LIN {X 0,Y 159.635,Z 839.585,A -85,B 0,C 180,E1 -24712.11,E2 -24712.11} C_VEL
LIN {X 0,Y 158.512,Z 849.666,A -85,B 0,C 180,E1 -24712.886,E2 -24712.886} C_VEL
LIN {X 0,Y 156.369,Z 861.365,A -85,B 0,C 180,E1 -24714.248,E2 -24714.248} C_VEL
LIN {X 0,Y 154.242,Z 870.146,A -85,B 0,C 180,E1 -24715.676,E2 -24715.676} C_VEL
LIN {X 0,Y 151.874,Z 878.505,A -85,B 0,C 180,E1 -24717.456,E2 -24717.456} C_VEL
LIN {X 0,Y 149.469,Z 885.387,A -85,B 0,C 180,E1 -24719.247,E2 -24719.247} C_VEL
LIN {X 0,Y 146.966,Z 892.073,A -85,B 0,C 180,E1 -24721.432,E2 -24721.432} C_VEL
LIN {X 0,Y 144.263,Z 898.407,A -85,B 0,C 180,E1 -24723.995,E2 -24723.995} C_VEL
LIN {X 0,Y 141.947,Z 903.667,A -85,B 0,C 180,E1 -24726.666,E2 -24726.666} C_VEL
LIN {X 0,Y 139.836,Z 908.059,A -85,B 0,C 180,E1 -24729.402,E2 -24729.402} C_VEL
LIN {X 0,Y 137.318,Z 913.221,A -85,B 0,C 180,E1 -24733.651,E2 -24733.651} C_VEL
LIN {X 0,Y 136.014,Z 915.865,A -85,B 0,C 180,E1 -24736.554,E2 -24736.554} C_VEL
LIN {X 0,Y 134.612,Z 918.759,A -85,B 0,C 180,E1 -24740.989,E2 -24740.989} C_VEL
LIN {X 0,Y 134.025,Z 920.018,A -85,B 0,C 180,E1 -24743.98,E2 -24743.98} C_VEL
LIN {X 0,Y 133.644,Z 920.881,A -85,B 0,C 180,E1 -24747.665,E2 -24747.665} C_VEL
LIN {X 0,Y 133.579,Z 920.989,A -85,B 0,C 180,E1 -24751.506,E2 -24751.506} C_VEL
LIN {X 0,Y 134.025,Z 920.078,A -85,B 0,C 180,E1 -24756.02,E2 -24756.02} C_VEL
LIN {X 0,Y 134.605,Z 918.859,A -85,B 0,C 180,E1 -24759.012,E2 -24759.012} C_VEL
LIN {X 0,Y 135.974,Z 916.007,A -85,B 0,C 180,E1 -24763.45,E2 -24763.45} C_VEL
LIN {X 0,Y 137.259,Z 913.408,A -85,B 0,C 180,E1 -24766.356,E2 -24766.356} C_VEL
LIN {X 0,Y 139.777,Z 908.296,A -85,B 0,C 180,E1 -24770.607,E2 -24770.607} C_VEL
LIN {X 0,Y 142.479,Z 902.79,A -85,B 0,C 180,E1 -24774.013,E2 -24774.013} C_VEL
LIN {X 0,Y 145.543,Z 895.866,A -85,B 0,C 180,E1 -24777.306,E2 -24777.306} C_VEL
LIN {X 0,Y 148.7,Z 887.912,A -85,B 0,C 180,E1 -24780.144,E2 -24780.144} C_VEL
LIN {X 0,Y 151.398,Z 880.327,A -85,B 0,C 180,E1 -24782.265,E2 -24782.265} C_VEL
LIN {X 0,Y 153.812,Z 872.37,A -85,B 0,C 180,E1 -24784.037,E2 -24784.037} C_VEL
LIN {X 0,Y 155.916,Z 864.14,A -85,B 0,C 180,E1 -24785.475,E2 -24785.475} C_VEL
LIN {X 0,Y 157.792,Z 855.078,A -85,B 0,C 180,E1 -24786.679,E2 -24786.679} C_VEL
LIN {X 0,Y 159.073,Z 846.352,A -85,B 0,C 180,E1 -24787.55,E2 -24787.55} C_VEL
LIN {X 0,Y 159.964,Z 837.426,A -85,B 0,C 180,E1 -24788.159,E2 -24788.159} C_VEL
LIN {X 0,Y 161.274,Z 812.923,A -85,B 0,C 180,E1 -24789.231,E2 -24789.231} C_VEL
LIN {X 0,Y 158.219,Z 805.845,A -85,B 0,C 180,E1 -24790.561,E2 -24790.561} C_VEL
LIN {X 0,Y 151.819,Z 794.198,A -85,B 0,C 180,E1 -24793.417,E2 -24793.417} C_VEL
LIN {X 0,Y 146.722,Z 786.269,A -85,B 0,C 180,E1 -24795.889,E2 -24795.889} C_VEL
LIN {X 0,Y 144.688,Z 783.348,A -85,B 0,C 180,E1 -24796.94,E2 -24796.94} C_VEL
LIN {X 0,Y 142.122,Z 779.603,A -85,B 0,C 180,E1 -24798.345,E2 -24798.345} C_VEL
LIN {X 0,Y 139.81,Z 776.247,A -85,B 0,C 180,E1 -24799.69,E2 -24799.69} C_VEL
LIN {X 0,Y 139.073,Z 775.314,A -85,B 0,C 180,E1 -24800.125,E2 -24800.125} C_VEL
LIN {X 0,Y 136.97,Z 773.087,A -85,B 0,C 180,E1 -24801.381,E2 -24801.381} C_VEL
LIN {X 0,Y 136.153,Z 770.959,A -85,B 0,C 180,E1 -24802.195,E2 -24802.195} C_VEL
LIN {X 0,Y 136.027,Z 770.381,A -85,B 0,C 180,E1 -24803.085,E2 -24803.085} C_VEL
LIN {X 0,Y 136.063,Z 770.334,A -85,B 0,C 180,E1 -24808.9,E2 -24808.9} C_VEL
LIN {X 0,Y 136.145,Z 770.314,A -85,B 0,C 180,E1 -24812.316,E2 -24812.316} C_VEL
LIN {X 0,Y 136.243,Z 770.325,A -85,B 0,C 180,E1 -24818.832,E2 -24818.832} C_VEL
LIN {X 0,Y 136.264,Z 770.295,A -85,B 0,C 180,E1 -24825.055,E2 -24825.055} C_VEL
LIN {X 0,Y 136.498,Z 770.293,A -85,B 0,C 180,E1 -24828.114,E2 -24828.114} C_VEL
LIN {X 0,Y 136.596,Z 770.241,A -85,B 0,C 180,E1 -24831.12,E2 -24831.12} C_VEL
LIN {X 0,Y 137.135,Z 770.182,A -85,B 0,C 180,E1 -24840,E2 -24840} C_VEL
LIN {X 0,Y 136.59,Z 770.268,A -85,B 0,C 180,E1 -24848.879,E2 -24848.879} C_VEL
LIN {X 0,Y 136.492,Z 770.252,A -85,B 0,C 180,E1 -24851.954,E2 -24851.954} C_VEL
LIN {X 0,Y 136.252,Z 770.315,A -85,B 0,C 180,E1 -24858.028,E2 -24858.028} C_VEL
LIN {X 0,Y 136.199,Z 770.294,A -85,B 0,C 180,E1 -24861.749,E2 -24861.749} C_VEL
LIN {X 0,Y 136.1,Z 770.315,A -85,B 0,C 180,E1 -24868.615,E2 -24868.615} C_VEL
LIN {X 0,Y 136.072,Z 770.314,A -85,B 0,C 180,E1 -24874.62,E2 -24874.62} C_VEL
LIN {X 0,Y 136.069,Z 770.603,A -85,B 0,C 180,E1 -24877.074,E2 -24877.074} C_VEL
LIN {X 0,Y 136.331,Z 771.59,A -85,B 0,C 180,E1 -24877.746,E2 -24877.746} C_VEL
LIN {X 0,Y 137.768,Z 774.133,A -85,B 0,C 180,E1 -24878.751,E2 -24878.751} C_VEL
LIN {X 0,Y 139.692,Z 775.951,A -85,B 0,C 180,E1 -24879.861,E2 -24879.861} C_VEL
LIN {X 0,Y 141.889,Z 779.358,A -85,B 0,C 180,E1 -24881.161,E2 -24881.161} C_VEL
LIN {X 0,Y 143.184,Z 781.06,A -85,B 0,C 180,E1 -24881.872,E2 -24881.872} C_VEL
LIN {X 0,Y 146.021,Z 785.342,A -85,B 0,C 180,E1 -24883.391,E2 -24883.391} C_VEL
LIN {X 0,Y 150.796,Z 794.191,A -85,B 0,C 180,E1 -24885.843,E2 -24885.843} C_VEL
LIN {X 0,Y 155.885,Z 805.497,A -85,B 0,C 180,E1 -24888.306,E2 -24888.306} C_VEL
LIN {X 0,Y 159.778,Z 815.797,A -85,B 0,C 180,E1 -24890.122,E2 -24890.122} C_VEL
LIN {X 0,Y 160.657,Z 825.932,A -85,B 0,C 180,E1 -24890.954,E2 -24890.954} C_VEL
LIN {X 0,Y 159.375,Z 846.828,A -85,B 0,C 180,E1 -24891.876,E2 -24891.876} C_VEL
LIN {X 0,Y 157.91,Z 858.37,A -85,B 0,C 180,E1 -24892.735,E2 -24892.735} C_VEL
LIN {X 0,Y 155.604,Z 869.497,A -85,B 0,C 180,E1 -24894.044,E2 -24894.044} C_VEL
LIN {X 0,Y 153.331,Z 878.512,A -85,B 0,C 180,E1 -24895.535,E2 -24895.535} C_VEL
LIN {X 0,Y 150.925,Z 886.424,A -85,B 0,C 180,E1 -24897.215,E2 -24897.215} C_VEL
LIN {X 0,Y 148.126,Z 894.308,A -85,B 0,C 180,E1 -24899.333,E2 -24899.333} C_VEL
LIN {X 0,Y 145.178,Z 901.651,A -85,B 0,C 180,E1 -24901.836,E2 -24901.836} C_VEL
LIN {X 0,Y 141.973,Z 909.104,A -85,B 0,C 180,E1 -24905.117,E2 -24905.117} C_VEL
LIN {X 0,Y 139.22,Z 914.946,A -85,B 0,C 180,E1 -24908.532,E2 -24908.532} C_VEL
LIN {X 0,Y 137.076,Z 919.559,A -85,B 0,C 180,E1 -24912.084,E2 -24912.084} C_VEL
LIN {X 0,Y 135.739,Z 922.56,A -85,B 0,C 180,E1 -24914.996,E2 -24914.996} C_VEL
LIN {X 0,Y 134.718,Z 924.892,A -85,B 0,C 180,E1 -24917.955,E2 -24917.955} C_VEL
LIN {X 0,Y 133.989,Z 926.641,A -85,B 0,C 180,E1 -24920.947,E2 -24920.947} C_VEL
LIN {X 0,Y 133.631,Z 927.895,A -85,B 0,C 180,E1 -24923.962,E2 -24923.962} C_VEL
LIN {X 0,Y 133.47,Z 928.674,A -85,B 0,C 180,E1 -24926.982,E2 -24926.982} C_VEL
LIN {X 0,Y 133.531,Z 928.971,A -85,B 0,C 180,E1 -24930,E2 -24930} C_VEL
LIN {X 0,Y 133.467,Z 928.664,A -85,B 0,C 180,E1 -24933.018,E2 -24933.018} C_VEL
LIN {X 0,Y 133.571,Z 927.863,A -85,B 0,C 180,E1 -24936.041,E2 -24936.041} C_VEL
LIN {X 0,Y 133.989,Z 926.589,A -85,B 0,C 180,E1 -24939.053,E2 -24939.053} C_VEL
LIN {X 0,Y 135.186,Z 923.659,A -85,B 0,C 180,E1 -24943.529,E2 -24943.529} C_VEL
LIN {X 0,Y 136.362,Z 920.99,A -85,B 0,C 180,E1 -24946.467,E2 -24946.467} C_VEL
LIN {X 0,Y 138.728,Z 915.782,A -85,B 0,C 180,E1 -24950.77,E2 -24950.77} C_VEL
LIN {X 0,Y 141.96,Z 908.923,A -85,B 0,C 180,E1 -24954.886,E2 -24954.886} C_VEL
LIN {X 0,Y 145.158,Z 901.434,A -85,B 0,C 180,E1 -24958.168,E2 -24958.168} C_VEL
LIN {X 0,Y 148.13,Z 894.053,A -85,B 0,C 180,E1 -24960.666,E2 -24960.666} C_VEL
LIN {X 0,Y 148.755,Z 892.384,A -85,B 0,C 180,E1 -24961.166,E2 -24961.166} C_VEL
LIN {X 0,Y 149.828,Z 887.833,A -85,B 0,C 180,E1 -24962.562,E2 -24962.562} C_VEL
LIN {X 0,Y 149.907,Z 880.057,A -85,B 0,C 180,E1 -24964.93,E2 -24964.93} C_VEL
LIN {X 0,Y 149.788,Z 871.747,A -85,B 0,C 180,E1 -24967.002,E2 -24967.002} C_VEL
LIN {X 0,Y 150.487,Z 866.362,A -85,B 0,C 180,E1 -24967.892,E2 -24967.892} C_VEL
LIN {X 0,Y 152.584,Z 855.455,A -85,B 0,C 180,E1 -24969.045,E2 -24969.045} C_VEL
LIN {X 0,Y 153.775,Z 846.031,A -85,B 0,C 180,E1 -24969.717,E2 -24969.717} C_VEL
LIN {X 0,Y 154.965,Z 825.846,A -85,B 0,C 180,E1 -24970.654,E2 -24970.654} C_VEL
LIN {X 0,Y 154.102,Z 817.408,A -85,B 0,C 180,E1 -24971.438,E2 -24971.438} C_VEL
LIN {X 0,Y 149.667,Z 805.878,A -85,B 0,C 180,E1 -24973.685,E2 -24973.685} C_VEL
LIN {X 0,Y 145.152,Z 796.052,A -85,B 0,C 180,E1 -24976.078,E2 -24976.078} C_VEL
LIN {X 0,Y 141.174,Z 788.802,A -85,B 0,C 180,E1 -24978.304,E2 -24978.304} C_VEL
LIN {X 0,Y 138.212,Z 784.573,A -85,B 0,C 180,E1 -24980.023,E2 -24980.023} C_VEL
LIN {X 0,Y 135.846,Z 781.103,A -85,B 0,C 180,E1 -24981.505,E2 -24981.505} C_VEL
LIN {X 0,Y 133.439,Z 778.063,A -85,B 0,C 180,E1 -24983.077,E2 -24983.077} C_VEL
LIN {X 0,Y 132.663,Z 776.576,A -85,B 0,C 180,E1 -24983.653,E2 -24983.653} C_VEL
LIN {X 0,Y 130.343,Z 774.52,A -85,B 0,C 180,E1 -24985.244,E2 -24985.244} C_VEL
LIN {X 0,Y 129.107,Z 771.819,A -85,B 0,C 180,E1 -24986.543,E2 -24986.543} C_VEL
LIN {X 0,Y 128.986,Z 771.241,A -85,B 0,C 180,E1 -24987.911,E2 -24987.911} C_VEL
LIN {X 0,Y 129.017,Z 771.195,A -85,B 0,C 180,E1 -24990.643,E2 -24990.643} C_VEL
LIN {X 0,Y 129.031,Z 771.225,A -85,B 0,C 180,E1 -24994.168,E2 -24994.168} C_VEL
LIN {X 0,Y 129.108,Z 771.178,A -85,B 0,C 180,E1 -24997.728,E2 -24997.728} C_VEL
LIN {X 0,Y 129.159,Z 771.183,A -85,B 0,C 180,E1 -25000.945,E2 -25000.945} C_VEL
LIN {X 0,Y 129.417,Z 771.132,A -85,B 0,C 180,E1 -25007.821,E2 -25007.821} C_VEL
LIN {X 0,Y 129.516,Z 771.14,A -85,B 0,C 180,E1 -25010.631,E2 -25010.631} C_VEL
LIN {X 0,Y 130.091,Z 771.058,A -85,B 0,C 180,E1 -25020,E2 -25020} C_VEL
LIN {X 0,Y 129.511,Z 771.125,A -85,B 0,C 180,E1 -25029.37,E2 -25029.37} C_VEL
LIN {X 0,Y 129.392,Z 771.181,A -85,B 0,C 180,E1 -25032.549,E2 -25032.549} C_VEL
LIN {X 0,Y 129.114,Z 771.181,A -85,B 0,C 180,E1 -25039.063,E2 -25039.063} C_VEL
LIN {X 0,Y 129.107,Z 771.209,A -85,B 0,C 180,E1 -25042.399,E2 -25042.399} C_VEL
LIN {X 0,Y 129.027,Z 771.19,A -85,B 0,C 180,E1 -25045.834,E2 -25045.834} C_VEL
LIN {X 0,Y 129.017,Z 771.221,A -85,B 0,C 180,E1 -25049.358,E2 -25049.358} C_VEL
LIN {X 0,Y 129.033,Z 771.485,A -85,B 0,C 180,E1 -25053.534,E2 -25053.534} C_VEL
LIN {X 0,Y 129.324,Z 772.589,A -85,B 0,C 180,E1 -25054.339,E2 -25054.339} C_VEL
LIN {X 0,Y 130.811,Z 775.152,A -85,B 0,C 180,E1 -25055.566,E2 -25055.566} C_VEL
LIN {X 0,Y 132.899,Z 777.009,A -85,B 0,C 180,E1 -25056.981,E2 -25056.981} C_VEL
LIN {X 0,Y 134.985,Z 780.287,A -85,B 0,C 180,E1 -25058.428,E2 -25058.428} C_VEL
LIN {X 0,Y 136.568,Z 782.116,A -85,B 0,C 180,E1 -25059.413,E2 -25059.413} C_VEL
LIN {X 0,Y 140.219,Z 787.446,A -85,B 0,C 180,E1 -25061.616,E2 -25061.616} C_VEL
LIN {X 0,Y 145.335,Z 795.26,A -85,B 0,C 180,E1 -25064.401,E2 -25064.401} C_VEL
LIN {X 0,Y 150.635,Z 804.437,A -85,B 0,C 180,E1 -25067.03,E2 -25067.03} C_VEL
LIN {X 0,Y 155.264,Z 813.871,A -85,B 0,C 180,E1 -25069.183,E2 -25069.183} C_VEL
LIN {X 0,Y 155.734,Z 815.756,A -85,B 0,C 180,E1 -25069.446,E2 -25069.446} C_VEL
LIN {X 0,Y 154.175,Z 838.958,A -85,B 0,C 180,E1 -25070.444,E2 -25070.444} C_VEL
LIN {X 0,Y 153.149,Z 848.227,A -85,B 0,C 180,E1 -25071.142,E2 -25071.142} C_VEL
LIN {X 0,Y 151.218,Z 859.169,A -85,B 0,C 180,E1 -25072.327,E2 -25072.327} C_VEL
LIN {X 0,Y 148.44,Z 870.36,A -85,B 0,C 180,E1 -25074.133,E2 -25074.133} C_VEL
LIN {X 0,Y 145.938,Z 878.718,A -85,B 0,C 180,E1 -25075.956,E2 -25075.956} C_VEL
LIN {X 0,Y 143.431,Z 885.598,A -85,B 0,C 180,E1 -25077.801,E2 -25077.801} C_VEL
LIN {X 0,Y 140.791,Z 892.284,A -85,B 0,C 180,E1 -25080.054,E2 -25080.054} C_VEL
LIN {X 0,Y 137.919,Z 898.618,A -85,B 0,C 180,E1 -25082.702,E2 -25082.702} C_VEL
LIN {X 0,Y 135.455,Z 903.878,A -85,B 0,C 180,E1 -25085.476,E2 -25085.476} C_VEL
LIN {X 0,Y 133.214,Z 908.269,A -85,B 0,C 180,E1 -25088.327,E2 -25088.327} C_VEL
LIN {X 0,Y 130.531,Z 913.431,A -85,B 0,C 180,E1 -25092.775,E2 -25092.775} C_VEL
LIN {X 0,Y 129.118,Z 916.075,A -85,B 0,C 180,E1 -25095.822,E2 -25095.822} C_VEL
LIN {X 0,Y 127.614,Z 918.969,A -85,B 0,C 180,E1 -25100.49,E2 -25100.49} C_VEL
LIN {X 0,Y 126.971,Z 920.228,A -85,B 0,C 180,E1 -25103.644,E2 -25103.644} C_VEL
LIN {X 0,Y 126.617,Z 921.018,A -85,B 0,C 180,E1 -25106.818,E2 -25106.818} C_VEL
LIN {X 0,Y 126.505,Z 921.319,A -85,B 0,C 180,E1 -25110,E2 -25110} C_VEL
LIN {X 0,Y 126.586,Z 921.039,A -85,B 0,C 180,E1 -25113.183,E2 -25113.183} C_VEL
LIN {X 0,Y 126.971,Z 920.286,A -85,B 0,C 180,E1 -25116.356,E2 -25116.356} C_VEL
LIN {X 0,Y 127.607,Z 919.068,A -85,B 0,C 180,E1 -25119.51,E2 -25119.51} C_VEL
LIN {X 0,Y 129.08,Z 916.215,A -85,B 0,C 180,E1 -25124.183,E2 -25124.183} C_VEL
LIN {X 0,Y 130.464,Z 913.616,A -85,B 0,C 180,E1 -25127.234,E2 -25127.234} C_VEL
LIN {X 0,Y 133.16,Z 908.503,A -85,B 0,C 180,E1 -25131.682,E2 -25131.682} C_VEL
LIN {X 0,Y 136.034,Z 902.997,A -85,B 0,C 180,E1 -25135.228,E2 -25135.228} C_VEL
LIN {X 0,Y 139.279,Z 896.072,A -85,B 0,C 180,E1 -25138.644,E2 -25138.644} C_VEL
LIN {X 0,Y 142.625,Z 888.117,A -85,B 0,C 180,E1 -25141.571,E2 -25141.571} C_VEL
LIN {X 0,Y 145.454,Z 880.531,A -85,B 0,C 180,E1 -25143.756,E2 -25143.756} C_VEL
LIN {X 0,Y 147.993,Z 872.574,A -85,B 0,C 180,E1 -25145.573,E2 -25145.573} C_VEL
LIN {X 0,Y 150.213,Z 864.342,A -85,B 0,C 180,E1 -25147.041,E2 -25147.041} C_VEL
LIN {X 0,Y 152.093,Z 855.662,A -85,B 0,C 180,E1 -25148.228,E2 -25148.228} C_VEL
LIN {X 0,Y 153.43,Z 847.101,A -85,B 0,C 180,E1 -25149.118,E2 -25149.118} C_VEL
LIN {X 0,Y 154.342,Z 838.914,A -85,B 0,C 180,E1 -25149.711,E2 -25149.711} C_VEL
LIN {X 0,Y 155.748,Z 814.926,A -85,B 0,C 180,E1 -25150.803,E2 -25150.803} C_VEL
LIN {X 0,Y 152.296,Z 807.458,A -85,B 0,C 180,E1 -25152.408,E2 -25152.408} C_VEL
LIN {X 0,Y 146.671,Z 797.355,A -85,B 0,C 180,E1 -25155.148,E2 -25155.148} C_VEL
LIN {X 0,Y 141.36,Z 789.057,A -85,B 0,C 180,E1 -25157.985,E2 -25157.985} C_VEL
LIN {X 0,Y 138.426,Z 784.813,A -85,B 0,C 180,E1 -25159.694,E2 -25159.694} C_VEL
LIN {X 0,Y 135.842,Z 781.12,A -85,B 0,C 180,E1 -25161.312,E2 -25161.312} C_VEL
LIN {X 0,Y 133.487,Z 778.201,A -85,B 0,C 180,E1 -25162.855,E2 -25162.855} C_VEL
LIN {X 0,Y 132.477,Z 776.49,A -85,B 0,C 180,E1 -25163.593,E2 -25163.593} C_VEL
LIN {X 0,Y 130.277,Z 774.484,A -85,B 0,C 180,E1 -25165.126,E2 -25165.126} C_VEL
LIN {X 0,Y 129.1,Z 771.782,A -85,B 0,C 180,E1 -25166.427,E2 -25166.427} C_VEL
LIN {X 0,Y 128.974,Z 771.233,A -85,B 0,C 180,E1 -25167.908,E2 -25167.908} C_VEL
LIN {X 0,Y 129.035,Z 771.221,A -85,B 0,C 180,E1 -25170.646,E2 -25170.646} C_VEL
LIN {X 0,Y 129.109,Z 771.207,A -85,B 0,C 180,E1 -25177.601,E2 -25177.601} C_VEL
LIN {X 0,Y 129.181,Z 771.169,A -85,B 0,C 180,E1 -25184.215,E2 -25184.215} C_VEL
LIN {X 0,Y 129.418,Z 771.177,A -85,B 0,C 180,E1 -25187.82,E2 -25187.82} C_VEL
LIN {X 0,Y 129.521,Z 771.125,A -85,B 0,C 180,E1 -25190.631,E2 -25190.631} C_VEL
LIN {X 0,Y 130.09,Z 771.059,A -85,B 0,C 180,E1 -25200,E2 -25200} C_VEL
LIN {X 0,Y 129.516,Z 771.14,A -85,B 0,C 180,E1 -25209.369,E2 -25209.369} C_VEL
LIN {X 0,Y 129.394,Z 771.135,A -85,B 0,C 180,E1 -25212.548,E2 -25212.548} C_VEL
LIN {X 0,Y 129.159,Z 771.183,A -85,B 0,C 180,E1 -25219.055,E2 -25219.055} C_VEL
LIN {X 0,Y 129.109,Z 771.179,A -85,B 0,C 180,E1 -25222.398,E2 -25222.398} C_VEL
LIN {X 0,Y 129.031,Z 771.225,A -85,B 0,C 180,E1 -25225.832,E2 -25225.832} C_VEL
LIN {X 0,Y 129.005,Z 771.255,A -85,B 0,C 180,E1 -25232.084,E2 -25232.084} C_VEL
LIN {X 0,Y 129.106,Z 771.784,A -85,B 0,C 180,E1 -25233.219,E2 -25233.219} C_VEL
LIN {X 0,Y 130.539,Z 774.745,A -85,B 0,C 180,E1 -25234.696,E2 -25234.696} C_VEL
LIN {X 0,Y 132.96,Z 777.036,A -85,B 0,C 180,E1 -25236.37,E2 -25236.37} C_VEL
LIN {X 0,Y 135.035,Z 780.3,A -85,B 0,C 180,E1 -25237.818,E2 -25237.818} C_VEL
LIN {X 0,Y 136.493,Z 781.884,A -85,B 0,C 180,E1 -25238.725,E2 -25238.725} C_VEL
LIN {X 0,Y 141.953,Z 789.956,A -85,B 0,C 180,E1 -25241.979,E2 -25241.979} C_VEL
LIN {X 0,Y 146.684,Z 799.062,A -85,B 0,C 180,E1 -25244.605,E2 -25244.605} C_VEL
LIN {X 0,Y 151.302,Z 809.666,A -85,B 0,C 180,E1 -25247.016,E2 -25247.016} C_VEL
LIN {X 0,Y 154.496,Z 818.541,A -85,B 0,C 180,E1 -25248.642,E2 -25248.642} C_VEL
LIN {X 0,Y 155.11,Z 827.574,A -85,B 0,C 180,E1 -25249.381,E2 -25249.381} C_VEL
LIN {X 0,Y 153.784,Z 847.481,A -85,B 0,C 180,E1 -25250.292,E2 -25250.292} C_VEL
LIN {X 0,Y 151.988,Z 859.859,A -85,B 0,C 180,E1 -25251.294,E2 -25251.294} C_VEL
LIN {X 0,Y 149.66,Z 870.325,A -85,B 0,C 180,E1 -25252.609,E2 -25252.609} C_VEL
LIN {X 0,Y 147.452,Z 878.55,A -85,B 0,C 180,E1 -25254.02,E2 -25254.02} C_VEL
LIN {X 0,Y 144.745,Z 886.981,A -85,B 0,C 180,E1 -25255.885,E2 -25255.885} C_VEL
LIN {X 0,Y 141.667,Z 895.125,A -85,B 0,C 180,E1 -25258.19,E2 -25258.19} C_VEL
LIN {X 0,Y 138.291,Z 903.144,A -85,B 0,C 180,E1 -25261.132,E2 -25261.132} C_VEL
LIN {X 0,Y 134.927,Z 910.138,A -85,B 0,C 180,E1 -25264.55,E2 -25264.55} C_VEL
LIN {X 0,Y 132.095,Z 915.699,A -85,B 0,C 180,E1 -25268.135,E2 -25268.135} C_VEL
LIN {X 0,Y 129.548,Z 920.878,A -85,B 0,C 180,E1 -25272.64,E2 -25272.64} C_VEL
LIN {X 0,Y 127.759,Z 924.684,A -85,B 0,C 180,E1 -25277.289,E2 -25277.289} C_VEL
LIN {X 0,Y 126.968,Z 926.432,A -85,B 0,C 180,E1 -25280.441,E2 -25280.441} C_VEL
LIN {X 0,Y 126.564,Z 927.687,A -85,B 0,C 180,E1 -25283.624,E2 -25283.624} C_VEL
LIN {X 0,Y 126.383,Z 928.466,A -85,B 0,C 180,E1 -25286.812,E2 -25286.812} C_VEL
LIN {X 0,Y 126.445,Z 928.762,A -85,B 0,C 180,E1 -25290,E2 -25290} C_VEL
LIN {X 0,Y 126.379,Z 928.455,A -85,B 0,C 180,E1 -25293.188,E2 -25293.188} C_VEL
LIN {X 0,Y 126.522,Z 927.654,A -85,B 0,C 180,E1 -25296.378,E2 -25296.378} C_VEL
LIN {X 0,Y 126.968,Z 926.379,A -85,B 0,C 180,E1 -25299.559,E2 -25299.559} C_VEL
LIN {X 0,Y 128.266,Z 923.448,A -85,B 0,C 180,E1 -25304.274,E2 -25304.274} C_VEL
LIN {X 0,Y 129.547,Z 920.779,A -85,B 0,C 180,E1 -25307.36,E2 -25307.36} C_VEL
LIN {X 0,Y 132.095,Z 915.571,A -85,B 0,C 180,E1 -25311.866,E2 -25311.866} C_VEL
LIN {X 0,Y 135.55,Z 908.712,A -85,B 0,C 180,E1 -25316.149,E2 -25316.149} C_VEL
LIN {X 0,Y 138.924,Z 901.222,A -85,B 0,C 180,E1 -25319.554,E2 -25319.554} C_VEL
LIN {X 0,Y 142.075,Z 893.841,A -85,B 0,C 180,E1 -25322.125,E2 -25322.125} C_VEL
LIN {X 0,Y 144.886,Z 886.228,A -85,B 0,C 180,E1 -25324.225,E2 -25324.225} C_VEL
LIN {X 0,Y 147.537,Z 877.723,A -85,B 0,C 180,E1 -25326.077,E2 -25326.077} C_VEL
LIN {X 0,Y 150.295,Z 867.26,A -85,B 0,C 180,E1 -25327.78,E2 -25327.78} C_VEL
LIN {X 0,Y 150.487,Z 866.362,A -85,B 0,C 180,E1 -25327.892,E2 -25327.892} C_VEL
LIN {X 0,Y 151.182,Z 860.851,A -85,B 0,C 180,E1 -25328.681,E2 -25328.681} C_VEL
LIN {X 0,Y 150.397,Z 851.78,A -85,B 0,C 180,E1 -25330.191,E2 -25330.191} C_VEL
LIN {X 0,Y 149.185,Z 842.523,A -85,B 0,C 180,E1 -25331.487,E2 -25331.487} C_VEL
LIN {X 0,Y 149.093,Z 836.717,A -85,B 0,C 180,E1 -25331.915,E2 -25331.915} C_VEL
LIN {X 0,Y 149.543,Z 826.064,A -85,B 0,C 180,E1 -25332.434,E2 -25332.434} C_VEL
LIN {X 0,Y 149.04,Z 820.348,A -85,B 0,C 180,E1 -25332.976,E2 -25332.976} C_VEL
LIN {X 0,Y 144.912,Z 809.373,A -85,B 0,C 180,E1 -25335.253,E2 -25335.253} C_VEL
LIN {X 0,Y 140.789,Z 800.186,A -85,B 0,C 180,E1 -25337.632,E2 -25337.632} C_VEL
LIN {X 0,Y 137.451,Z 793.945,A -85,B 0,C 180,E1 -25339.656,E2 -25339.656} C_VEL
LIN {X 0,Y 134.408,Z 789.463,A -85,B 0,C 180,E1 -25341.569,E2 -25341.569} C_VEL
LIN {X 0,Y 132.393,Z 786.53,A -85,B 0,C 180,E1 -25342.93,E2 -25342.93} C_VEL
LIN {X 0,Y 129.981,Z 783.042,A -85,B 0,C 180,E1 -25344.672,E2 -25344.672} C_VEL
LIN {X 0,Y 127.067,Z 779.637,A -85,B 0,C 180,E1 -25346.895,E2 -25346.895} C_VEL
LIN {X 0,Y 125.849,Z 777.609,A -85,B 0,C 180,E1 -25347.959,E2 -25347.959} C_VEL
LIN {X 0,Y 123.301,Z 775.404,A -85,B 0,C 180,E1 -25350.136,E2 -25350.136} C_VEL
LIN {X 0,Y 122.033,Z 772.697,A -85,B 0,C 180,E1 -25351.811,E2 -25351.811} C_VEL
LIN {X 0,Y 121.956,Z 772.124,A -85,B 0,C 180,E1 -25353.474,E2 -25353.474} C_VEL
LIN {X 0,Y 122.029,Z 772.063,A -85,B 0,C 180,E1 -25357.145,E2 -25357.145} C_VEL
LIN {X 0,Y 122.116,Z 772.085,A -85,B 0,C 180,E1 -25363.277,E2 -25363.277} C_VEL
LIN {X 0,Y 122.364,Z 772.01,A -85,B 0,C 180,E1 -25367.527,E2 -25367.527} C_VEL
LIN {X 0,Y 122.446,Z 772.013,A -85,B 0,C 180,E1 -25370.085,E2 -25370.085} C_VEL
LIN {X 0,Y 122.604,Z 771.978,A -85,B 0,C 180,E1 -25376.714,E2 -25376.714} C_VEL
LIN {X 0,Y 123.044,Z 771.935,A -85,B 0,C 180,E1 -25380,E2 -25380} C_VEL
LIN {X 0,Y 122.419,Z 772.001,A -85,B 0,C 180,E1 -25387.089,E2 -25387.089} C_VEL
LIN {X 0,Y 122.364,Z 772.056,A -85,B 0,C 180,E1 -25392.472,E2 -25392.472} C_VEL
LIN {X 0,Y 122.021,Z 772.076,A -85,B 0,C 180,E1 -25400.218,E2 -25400.218} C_VEL
LIN {X 0,Y 121.982,Z 772.077,A -85,B 0,C 180,E1 -25403.785,E2 -25403.785} C_VEL
LIN {X 0,Y 121.977,Z 772.402,A -85,B 0,C 180,E1 -25408.266,E2 -25408.266} C_VEL
LIN {X 0,Y 122.347,Z 773.615,A -85,B 0,C 180,E1 -25409.294,E2 -25409.294} C_VEL
LIN {X 0,Y 123.736,Z 776.07,A -85,B 0,C 180,E1 -25410.743,E2 -25410.743} C_VEL
LIN {X 0,Y 126.182,Z 777.945,A -85,B 0,C 180,E1 -25412.773,E2 -25412.773} C_VEL
LIN {X 0,Y 128.034,Z 781.091,A -85,B 0,C 180,E1 -25414.359,E2 -25414.359} C_VEL
LIN {X 0,Y 130.016,Z 783.198,A -85,B 0,C 180,E1 -25415.823,E2 -25415.823} C_VEL
LIN {X 0,Y 132.485,Z 786.66,A -85,B 0,C 180,E1 -25417.593,E2 -25417.593} C_VEL
LIN {X 0,Y 136.466,Z 792.391,A -85,B 0,C 180,E1 -25420.193,E2 -25420.193} C_VEL
LIN {X 0,Y 142.6,Z 802.122,A -85,B 0,C 180,E1 -25423.752,E2 -25423.752} C_VEL
LIN {X 0,Y 148.357,Z 813.011,A -85,B 0,C 180,E1 -25426.761,E2 -25426.761} C_VEL
LIN {X 0,Y 150.218,Z 816.904,A -85,B 0,C 180,E1 -25427.678,E2 -25427.678} C_VEL
LIN {X 0,Y 148.687,Z 840.407,A -85,B 0,C 180,E1 -25428.78,E2 -25428.78} C_VEL
LIN {X 0,Y 147.161,Z 852.138,A -85,B 0,C 180,E1 -25429.768,E2 -25429.768} C_VEL
LIN {X 0,Y 145.108,Z 861.794,A -85,B 0,C 180,E1 -25430.977,E2 -25430.977} C_VEL
LIN {X 0,Y 142.757,Z 870.573,A -85,B 0,C 180,E1 -25432.466,E2 -25432.466} C_VEL
LIN {X 0,Y 140.12,Z 878.93,A -85,B 0,C 180,E1 -25434.333,E2 -25434.333} C_VEL
LIN {X 0,Y 137.491,Z 885.81,A -85,B 0,C 180,E1 -25436.228,E2 -25436.228} C_VEL
LIN {X 0,Y 134.698,Z 892.495,A -85,B 0,C 180,E1 -25438.55,E2 -25438.55} C_VEL
LIN {X 0,Y 131.655,Z 898.829,A -85,B 0,C 180,E1 -25441.286,E2 -25441.286} C_VEL
LIN {X 0,Y 129.029,Z 904.088,A -85,B 0,C 180,E1 -25444.167,E2 -25444.167} C_VEL
LIN {X 0,Y 126.647,Z 908.479,A -85,B 0,C 180,E1 -25447.142,E2 -25447.142} C_VEL
LIN {X 0,Y 123.769,Z 913.641,A -85,B 0,C 180,E1 -25451.802,E2 -25451.802} C_VEL
LIN {X 0,Y 122.255,Z 916.285,A -85,B 0,C 180,E1 -25455.008,E2 -25455.008} C_VEL
LIN {X 0,Y 120.617,Z 919.178,A -85,B 0,C 180,E1 -25459.933,E2 -25459.933} C_VEL
LIN {X 0,Y 119.916,Z 920.437,A -85,B 0,C 180,E1 -25463.269,E2 -25463.269} C_VEL
LIN {X 0,Y 119.54,Z 921.227,A -85,B 0,C 180,E1 -25466.63,E2 -25466.63} C_VEL
LIN {X 0,Y 119.419,Z 921.528,A -85,B 0,C 180,E1 -25470,E2 -25470} C_VEL
LIN {X 0,Y 119.5,Z 921.247,A -85,B 0,C 180,E1 -25473.372,E2 -25473.372} C_VEL
LIN {X 0,Y 119.916,Z 920.495,A -85,B 0,C 180,E1 -25476.731,E2 -25476.731} C_VEL
LIN {X 0,Y 120.61,Z 919.276,A -85,B 0,C 180,E1 -25480.068,E2 -25480.068} C_VEL
LIN {X 0,Y 122.221,Z 916.423,A -85,B 0,C 180,E1 -25484.997,E2 -25484.997} C_VEL
LIN {X 0,Y 123.699,Z 913.823,A -85,B 0,C 180,E1 -25488.209,E2 -25488.209} C_VEL
LIN {X 0,Y 126.601,Z 908.71,A -85,B 0,C 180,E1 -25492.867,E2 -25492.867} C_VEL
LIN {X 0,Y 129.652,Z 903.204,A -85,B 0,C 180,E1 -25496.565,E2 -25496.565} C_VEL
LIN {X 0,Y 133.099,Z 896.278,A -85,B 0,C 180,E1 -25500.108,E2 -25500.108} C_VEL
LIN {X 0,Y 136.633,Z 888.323,A -85,B 0,C 180,E1 -25503.129,E2 -25503.129} C_VEL
LIN {X 0,Y 139.609,Z 880.736,A -85,B 0,C 180,E1 -25505.374,E2 -25505.374} C_VEL
LIN {X 0,Y 142.29,Z 872.777,A -85,B 0,C 180,E1 -25507.233,E2 -25507.233} C_VEL
LIN {X 0,Y 144.625,Z 864.544,A -85,B 0,C 180,E1 -25508.73,E2 -25508.73} C_VEL
LIN {X 0,Y 146.527,Z 856.163,A -85,B 0,C 180,E1 -25509.908,E2 -25509.908} C_VEL
LIN {X 0,Y 148.004,Z 847.266,A -85,B 0,C 180,E1 -25510.852,E2 -25510.852} C_VEL
LIN {X 0,Y 148.959,Z 839.107,A -85,B 0,C 180,E1 -25511.453,E2 -25511.453} C_VEL
LIN {X 0,Y 150.364,Z 817.143,A -85,B 0,C 180,E1 -25512.469,E2 -25512.469} C_VEL
LIN {X 0,Y 145.323,Z 806.897,A -85,B 0,C 180,E1 -25515.028,E2 -25515.028} C_VEL
LIN {X 0,Y 139.495,Z 796.988,A -85,B 0,C 180,E1 -25518.242,E2 -25518.242} C_VEL
LIN {X 0,Y 134.973,Z 790.201,A -85,B 0,C 180,E1 -25521.016,E2 -25521.016} C_VEL
LIN {X 0,Y 132.603,Z 786.76,A -85,B 0,C 180,E1 -25522.609,E2 -25522.609} C_VEL
LIN {X 0,Y 130.135,Z 783.36,A -85,B 0,C 180,E1 -25524.38,E2 -25524.38} C_VEL
LIN {X 0,Y 129.36,Z 782.368,A -85,B 0,C 180,E1 -25524.959,E2 -25524.959} C_VEL
LIN {X 0,Y 127.038,Z 779.658,A -85,B 0,C 180,E1 -25526.767,E2 -25526.767} C_VEL
LIN {X 0,Y 125.944,Z 777.662,A -85,B 0,C 180,E1 -25527.75,E2 -25527.75} C_VEL
LIN {X 0,Y 123.351,Z 775.485,A -85,B 0,C 180,E1 -25529.975,E2 -25529.975} C_VEL
LIN {X 0,Y 122.051,Z 772.712,A -85,B 0,C 180,E1 -25531.658,E2 -25531.658} C_VEL
LIN {X 0,Y 121.953,Z 772.111,A -85,B 0,C 180,E1 -25533.01,E2 -25533.01} C_VEL
LIN {X 0,Y 122.023,Z 772.082,A -85,B 0,C 180,E1 -25537.151,E2 -25537.151} C_VEL
LIN {X 0,Y 122.093,Z 772.047,A -85,B 0,C 180,E1 -25543.273,E2 -25543.273} C_VEL
LIN {X 0,Y 122.365,Z 772.056,A -85,B 0,C 180,E1 -25547.526,E2 -25547.526} C_VEL
LIN {X 0,Y 122.45,Z 772.01,A -85,B 0,C 180,E1 -25550.085,E2 -25550.085} C_VEL
LIN {X 0,Y 122.627,Z 772.017,A -85,B 0,C 180,E1 -25556.714,E2 -25556.714} C_VEL
LIN {X 0,Y 123.044,Z 771.935,A -85,B 0,C 180,E1 -25560,E2 -25560} C_VEL
LIN {X 0,Y 122.446,Z 772.038,A -85,B 0,C 180,E1 -25566.591,E2 -25566.591} C_VEL
LIN {X 0,Y 122.446,Z 772.012,A -85,B 0,C 180,E1 -25569.915,E2 -25569.915} C_VEL
LIN {X 0,Y 122.264,Z 772.025,A -85,B 0,C 180,E1 -25573.292,E2 -25573.292} C_VEL
LIN {X 0,Y 122.048,Z 772.058,A -85,B 0,C 180,E1 -25580.212,E2 -25580.212} C_VEL
LIN {X 0,Y 121.989,Z 772.103,A -85,B 0,C 180,E1 -25585.6,E2 -25585.6} C_VEL
LIN {X 0,Y 121.978,Z 772.462,A -85,B 0,C 180,E1 -25587.598,E2 -25587.598} C_VEL
LIN {X 0,Y 122.383,Z 773.815,A -85,B 0,C 180,E1 -25588.632,E2 -25588.632} C_VEL
LIN {X 0,Y 124.215,Z 776.403,A -85,B 0,C 180,E1 -25590.446,E2 -25590.446} C_VEL
LIN {X 0,Y 126.265,Z 778.085,A -85,B 0,C 180,E1 -25592.158,E2 -25592.158} C_VEL
LIN {X 0,Y 128.462,Z 781.519,A -85,B 0,C 180,E1 -25594.01,E2 -25594.01} C_VEL
LIN {X 0,Y 130.063,Z 783.155,A -85,B 0,C 180,E1 -25595.187,E2 -25595.187} C_VEL
LIN {X 0,Y 132.717,Z 786.88,A -85,B 0,C 180,E1 -25597.098,E2 -25597.098} C_VEL
LIN {X 0,Y 138.16,Z 794.893,A -85,B 0,C 180,E1 -25600.598,E2 -25600.598} C_VEL
LIN {X 0,Y 143.146,Z 804.915,A -85,B 0,C 180,E1 -25603.577,E2 -25603.577} C_VEL
LIN {X 0,Y 147.832,Z 816.698,A -85,B 0,C 180,E1 -25606.222,E2 -25606.222} C_VEL
LIN {X 0,Y 149.312,Z 821.288,A -85,B 0,C 180,E1 -25607.055,E2 -25607.055} C_VEL
LIN {X 0,Y 149.759,Z 828.198,A -85,B 0,C 180,E1 -25607.652,E2 -25607.652} C_VEL
LIN {X 0,Y 148.375,Z 847.514,A -85,B 0,C 180,E1 -25608.554,E2 -25608.554} C_VEL
LIN {X 0,Y 146.41,Z 860.177,A -85,B 0,C 180,E1 -25609.62,E2 -25609.62} C_VEL
LIN {X 0,Y 144.364,Z 869.091,A -85,B 0,C 180,E1 -25610.738,E2 -25610.738} C_VEL
LIN {X 0,Y 141.946,Z 877.76,A -85,B 0,C 180,E1 -25612.214,E2 -25612.214} C_VEL
LIN {X 0,Y 139.447,Z 885.305,A -85,B 0,C 180,E1 -25613.865,E2 -25613.865} C_VEL
LIN {X 0,Y 136.525,Z 892.873,A -85,B 0,C 180,E1 -25615.957,E2 -25615.957} C_VEL
LIN {X 0,Y 133.603,Z 899.529,A -85,B 0,C 180,E1 -25618.262,E2 -25618.262} C_VEL
LIN {X 0,Y 130.608,Z 905.853,A -85,B 0,C 180,E1 -25621.034,E2 -25621.034} C_VEL
LIN {X 0,Y 127.894,Z 911.107,A -85,B 0,C 180,E1 -25623.921,E2 -25623.921} C_VEL
LIN {X 0,Y 125.519,Z 915.491,A -85,B 0,C 180,E1 -25626.925,E2 -25626.925} C_VEL
LIN {X 0,Y 122.772,Z 920.67,A -85,B 0,C 180,E1 -25631.649,E2 -25631.649} C_VEL
LIN {X 0,Y 120.828,Z 924.475,A -85,B 0,C 180,E1 -25636.546,E2 -25636.546} C_VEL
LIN {X 0,Y 119.97,Z 926.223,A -85,B 0,C 180,E1 -25639.878,E2 -25639.878} C_VEL
LIN {X 0,Y 119.492,Z 927.477,A -85,B 0,C 180,E1 -25643.245,E2 -25643.245} C_VEL
LIN {X 0,Y 119.291,Z 928.257,A -85,B 0,C 180,E1 -25646.622,E2 -25646.622} C_VEL
LIN {X 0,Y 119.36,Z 928.554,A -85,B 0,C 180,E1 -25650,E2 -25650} C_VEL
LIN {X 0,Y 119.288,Z 928.246,A -85,B 0,C 180,E1 -25653.378,E2 -25653.378} C_VEL
LIN {X 0,Y 119.462,Z 927.444,A -85,B 0,C 180,E1 -25656.757,E2 -25656.757} C_VEL
LIN {X 0,Y 119.97,Z 926.169,A -85,B 0,C 180,E1 -25660.122,E2 -25660.122} C_VEL
LIN {X 0,Y 121.37,Z 923.237,A -85,B 0,C 180,E1 -25665.104,E2 -25665.104} C_VEL
LIN {X 0,Y 122.771,Z 920.569,A -85,B 0,C 180,E1 -25668.352,E2 -25668.352} C_VEL
LIN {X 0,Y 125.518,Z 915.36,A -85,B 0,C 180,E1 -25673.076,E2 -25673.076} C_VEL
LIN {X 0,Y 129.215,Z 908.501,A -85,B 0,C 180,E1 -25677.537,E2 -25677.537} C_VEL
LIN {X 0,Y 132.788,Z 901.011,A -85,B 0,C 180,E1 -25681.067,E2 -25681.067} C_VEL
LIN {X 0,Y 136.11,Z 893.629,A -85,B 0,C 180,E1 -25683.716,E2 -25683.716} C_VEL
LIN {X 0,Y 139.083,Z 885.959,A -85,B 0,C 180,E1 -25685.887,E2 -25685.887} C_VEL
LIN {X 0,Y 141.913,Z 877.355,A -85,B 0,C 180,E1 -25687.796,E2 -25687.796} C_VEL
LIN {X 0,Y 144.857,Z 866.555,A -85,B 0,C 180,E1 -25689.564,E2 -25689.564} C_VEL
LIN {X 0,Y 147.117,Z 855.45,A -85,B 0,C 180,E1 -25690.764,E2 -25690.764} C_VEL
LIN {X 0,Y 148.328,Z 846.305,A -85,B 0,C 180,E1 -25691.445,E2 -25691.445} C_VEL
LIN {X 0,Y 149.093,Z 836.717,A -85,B 0,C 180,E1 -25691.915,E2 -25691.915} C_VEL
LIN {X 0,Y 148.846,Z 832.9,A -85,B 0,C 180,E1 -25692.242,E2 -25692.242} C_VEL
LIN {X 0,Y 147.833,Z 829.369,A -85,B 0,C 180,E1 -25692.825,E2 -25692.825} C_VEL
LIN {X 0,Y 142.519,Z 818.709,A -85,B 0,C 180,E1 -25695.565,E2 -25695.565} C_VEL
LIN {X 0,Y 138.36,Z 808.18,A -85,B 0,C 180,E1 -25698.128,E2 -25698.128} C_VEL
LIN {X 0,Y 134.184,Z 799.574,A -85,B 0,C 180,E1 -25700.846,E2 -25700.846} C_VEL
LIN {X 0,Y 129.384,Z 792.311,A -85,B 0,C 180,E1 -25704.178,E2 -25704.178} C_VEL
LIN {X 0,Y 126.41,Z 788.211,A -85,B 0,C 180,E1 -25706.481,E2 -25706.481} C_VEL
LIN {X 0,Y 123.859,Z 784.704,A -85,B 0,C 180,E1 -25708.669,E2 -25708.669} C_VEL
LIN {X 0,Y 123.051,Z 783.672,A -85,B 0,C 180,E1 -25709.403,E2 -25709.403} C_VEL
LIN {X 0,Y 120.583,Z 781.038,A -85,B 0,C 180,E1 -25711.748,E2 -25711.748} C_VEL
LIN {X 0,Y 119.404,Z 778.795,A -85,B 0,C 180,E1 -25713.098,E2 -25713.098} C_VEL
LIN {X 0,Y 116.574,Z 776.667,A -85,B 0,C 180,E1 -25716.266,E2 -25716.266} C_VEL
LIN {X 0,Y 115.1,Z 773.682,A -85,B 0,C 180,E1 -25718.744,E2 -25718.744} C_VEL
LIN {X 0,Y 114.995,Z 773.009,A -85,B 0,C 180,E1 -25720.359,E2 -25720.359} C_VEL
LIN {X 0,Y 115.285,Z 772.891,A -85,B 0,C 180,E1 -25727.263,E2 -25727.263} C_VEL
LIN {X 0,Y 115.388,Z 772.921,A -85,B 0,C 180,E1 -25733.004,E2 -25733.004} C_VEL
LIN {X 0,Y 115.996,Z 772.811,A -85,B 0,C 180,E1 -25740,E2 -25740} C_VEL
LIN {X 0,Y 115.387,Z 772.877,A -85,B 0,C 180,E1 -25746.997,E2 -25746.997} C_VEL
LIN {X 0,Y 115.285,Z 772.937,A -85,B 0,C 180,E1 -25752.736,E2 -25752.736} C_VEL
LIN {X 0,Y 115.008,Z 773.114,A -85,B 0,C 180,E1 -25760.572,E2 -25760.572} C_VEL
LIN {X 0,Y 115.195,Z 774.074,A -85,B 0,C 180,E1 -25762.071,E2 -25762.071} C_VEL
LIN {X 0,Y 116.901,Z 777.108,A -85,B 0,C 180,E1 -25764.615,E2 -25764.615} C_VEL
LIN {X 0,Y 119.587,Z 779.079,A -85,B 0,C 180,E1 -25767.569,E2 -25767.569} C_VEL
LIN {X 0,Y 121.276,Z 782.133,A -85,B 0,C 180,E1 -25769.439,E2 -25769.439} C_VEL
LIN {X 0,Y 123.749,Z 784.556,A -85,B 0,C 180,E1 -25771.691,E2 -25771.691} C_VEL
LIN {X 0,Y 126.116,Z 787.915,A -85,B 0,C 180,E1 -25773.747,E2 -25773.747} C_VEL
LIN {X 0,Y 127.313,Z 789.442,A -85,B 0,C 180,E1 -25774.701,E2 -25774.701} C_VEL
LIN {X 0,Y 130.864,Z 794.55,A -85,B 0,C 180,E1 -25777.362,E2 -25777.362} C_VEL
LIN {X 0,Y 135.265,Z 801.291,A -85,B 0,C 180,E1 -25780.306,E2 -25780.306} C_VEL
LIN {X 0,Y 140.345,Z 810.081,A -85,B 0,C 180,E1 -25783.36,E2 -25783.36} C_VEL
LIN {X 0,Y 144.913,Z 819.302,A -85,B 0,C 180,E1 -25785.884,E2 -25785.884} C_VEL
LIN {X 0,Y 143.42,Z 840.803,A -85,B 0,C 180,E1 -25786.926,E2 -25786.926} C_VEL
LIN {X 0,Y 141.679,Z 853.009,A -85,B 0,C 180,E1 -25787.992,E2 -25787.992} C_VEL
LIN {X 0,Y 139.664,Z 862.009,A -85,B 0,C 180,E1 -25789.143,E2 -25789.143} C_VEL
LIN {X 0,Y 137.183,Z 870.837,A -85,B 0,C 180,E1 -25790.671,E2 -25790.671} C_VEL
LIN {X 0,Y 134.428,Z 879.143,A -85,B 0,C 180,E1 -25792.572,E2 -25792.572} C_VEL
LIN {X 0,Y 131.652,Z 886.022,A -85,B 0,C 180,E1 -25794.511,E2 -25794.511} C_VEL
LIN {X 0,Y 128.707,Z 892.706,A -85,B 0,C 180,E1 -25796.904,E2 -25796.904} C_VEL
LIN {X 0,Y 125.484,Z 899.04,A -85,B 0,C 180,E1 -25799.731,E2 -25799.731} C_VEL
LIN {X 0,Y 122.679,Z 904.299,A -85,B 0,C 180,E1 -25802.722,E2 -25802.722} C_VEL
LIN {X 0,Y 120.145,Z 908.69,A -85,B 0,C 180,E1 -25805.828,E2 -25805.828} C_VEL
LIN {X 0,Y 117.043,Z 913.851,A -85,B 0,C 180,E1 -25810.716,E2 -25810.716} C_VEL
LIN {X 0,Y 115.43,Z 916.494,A -85,B 0,C 180,E1 -25814.098,E2 -25814.098} C_VEL
LIN {X 0,Y 113.651,Z 919.387,A -85,B 0,C 180,E1 -25819.309,E2 -25819.309} C_VEL
LIN {X 0,Y 112.875,Z 920.646,A -85,B 0,C 180,E1 -25822.847,E2 -25822.847} C_VEL
LIN {X 0,Y 112.471,Z 921.435,A -85,B 0,C 180,E1 -25826.417,E2 -25826.417} C_VEL
LIN {X 0,Y 112.335,Z 921.736,A -85,B 0,C 180,E1 -25830,E2 -25830} C_VEL
LIN {X 0,Y 112.427,Z 921.456,A -85,B 0,C 180,E1 -25833.584,E2 -25833.584} C_VEL
LIN {X 0,Y 112.874,Z 920.703,A -85,B 0,C 180,E1 -25837.153,E2 -25837.153} C_VEL
LIN {X 0,Y 113.644,Z 919.483,A -85,B 0,C 180,E1 -25840.692,E2 -25840.692} C_VEL
LIN {X 0,Y 115.372,Z 916.631,A -85,B 0,C 180,E1 -25845.91,E2 -25845.91} C_VEL
LIN {X 0,Y 116.98,Z 914.031,A -85,B 0,C 180,E1 -25849.295,E2 -25849.295} C_VEL
LIN {X 0,Y 120.105,Z 908.917,A -85,B 0,C 180,E1 -25854.18,E2 -25854.18} C_VEL
LIN {X 0,Y 123.349,Z 903.41,A -85,B 0,C 180,E1 -25858.038,E2 -25858.038} C_VEL
LIN {X 0,Y 127.02,Z 896.484,A -85,B 0,C 180,E1 -25861.711,E2 -25861.711} C_VEL
LIN {X 0,Y 130.753,Z 888.528,A -85,B 0,C 180,E1 -25864.827,E2 -25864.827} C_VEL
LIN {X 0,Y 133.888,Z 880.941,A -85,B 0,C 180,E1 -25867.132,E2 -25867.132} C_VEL
LIN {X 0,Y 136.697,Z 873.033,A -85,B 0,C 180,E1 -25869.019,E2 -25869.019} C_VEL
LIN {X 0,Y 138.991,Z 865.42,A -85,B 0,C 180,E1 -25870.447,E2 -25870.447} C_VEL
LIN {X 0,Y 141.079,Z 856.803,A -85,B 0,C 180,E1 -25871.697,E2 -25871.697} C_VEL
LIN {X 0,Y 142.601,Z 848.206,A -85,B 0,C 180,E1 -25872.65,E2 -25872.65} C_VEL
LIN {X 0,Y 143.742,Z 839.171,A -85,B 0,C 180,E1 -25873.329,E2 -25873.329} C_VEL
LIN {X 0,Y 145.035,Z 819.405,A -85,B 0,C 180,E1 -25874.287,E2 -25874.287} C_VEL
LIN {X 0,Y 139.775,Z 808.893,A -85,B 0,C 180,E1 -25877.22,E2 -25877.22} C_VEL
LIN {X 0,Y 134.335,Z 799.724,A -85,B 0,C 180,E1 -25880.561,E2 -25880.561} C_VEL
LIN {X 0,Y 129.622,Z 792.61,A -85,B 0,C 180,E1 -25883.837,E2 -25883.837} C_VEL
LIN {X 0,Y 126.515,Z 788.297,A -85,B 0,C 180,E1 -25886.254,E2 -25886.254} C_VEL
LIN {X 0,Y 124.109,Z 785.143,A -85,B 0,C 180,E1 -25888.307,E2 -25888.307} C_VEL
LIN {X 0,Y 123.24,Z 783.821,A -85,B 0,C 180,E1 -25889.12,E2 -25889.12} C_VEL
LIN {X 0,Y 120.755,Z 781.263,A -85,B 0,C 180,E1 -25891.48,E2 -25891.48} C_VEL
LIN {X 0,Y 119.355,Z 778.716,A -85,B 0,C 180,E1 -25893.085,E2 -25893.085} C_VEL
LIN {X 0,Y 116.561,Z 776.657,A -85,B 0,C 180,E1 -25896.266,E2 -25896.266} C_VEL
LIN {X 0,Y 115.063,Z 773.579,A -85,B 0,C 180,E1 -25898.97,E2 -25898.97} C_VEL
LIN {X 0,Y 114.979,Z 772.976,A -85,B 0,C 180,E1 -25901.282,E2 -25901.282} C_VEL
LIN {X 0,Y 115.286,Z 772.936,A -85,B 0,C 180,E1 -25907.261,E2 -25907.261} C_VEL
LIN {X 0,Y 115.393,Z 772.876,A -85,B 0,C 180,E1 -25913.003,E2 -25913.003} C_VEL
LIN {X 0,Y 115.996,Z 772.811,A -85,B 0,C 180,E1 -25920,E2 -25920} C_VEL
LIN {X 0,Y 115.388,Z 772.922,A -85,B 0,C 180,E1 -25926.996,E2 -25926.996} C_VEL
LIN {X 0,Y 115.285,Z 772.892,A -85,B 0,C 180,E1 -25932.737,E2 -25932.737} C_VEL
LIN {X 0,Y 115.045,Z 773.239,A -85,B 0,C 180,E1 -25940.098,E2 -25940.098} C_VEL
LIN {X 0,Y 115.302,Z 774.365,A -85,B 0,C 180,E1 -25941.451,E2 -25941.451} C_VEL
LIN {X 0,Y 117.085,Z 777.216,A -85,B 0,C 180,E1 -25944.03,E2 -25944.03} C_VEL
LIN {X 0,Y 119.537,Z 778.975,A -85,B 0,C 180,E1 -25946.752,E2 -25946.752} C_VEL
LIN {X 0,Y 121.642,Z 782.415,A -85,B 0,C 180,E1 -25949.052,E2 -25949.052} C_VEL
LIN {X 0,Y 123.755,Z 784.396,A -85,B 0,C 180,E1 -25950.974,E2 -25950.974} C_VEL
LIN {X 0,Y 126.195,Z 787.973,A -85,B 0,C 180,E1 -25953.125,E2 -25953.125} C_VEL
LIN {X 0,Y 127.428,Z 789.517,A -85,B 0,C 180,E1 -25954.111,E2 -25954.111} C_VEL
LIN {X 0,Y 130.965,Z 794.605,A -85,B 0,C 180,E1 -25956.775,E2 -25956.775} C_VEL
LIN {X 0,Y 134.562,Z 800.132,A -85,B 0,C 180,E1 -25959.222,E2 -25959.222} C_VEL
LIN {X 0,Y 139.069,Z 809.652,A -85,B 0,C 180,E1 -25962.151,E2 -25962.151} C_VEL
LIN {X 0,Y 143.398,Z 820.911,A -85,B 0,C 180,E1 -25964.803,E2 -25964.803} C_VEL
LIN {X 0,Y 144.192,Z 823.257,A -85,B 0,C 180,E1 -25965.279,E2 -25965.279} C_VEL
LIN {X 0,Y 144.5,Z 829.343,A -85,B 0,C 180,E1 -25965.812,E2 -25965.812} C_VEL
LIN {X 0,Y 143.135,Z 847.29,A -85,B 0,C 180,E1 -25966.672,E2 -25966.672} C_VEL
LIN {X 0,Y 141.377,Z 858.668,A -85,B 0,C 180,E1 -25967.604,E2 -25967.604} C_VEL
LIN {X 0,Y 138.93,Z 868.888,A -85,B 0,C 180,E1 -25968.881,E2 -25968.881} C_VEL
LIN {X 0,Y 136.406,Z 877.555,A -85,B 0,C 180,E1 -25970.387,E2 -25970.387} C_VEL
LIN {X 0,Y 133.372,Z 886.117,A -85,B 0,C 180,E1 -25972.331,E2 -25972.331} C_VEL
LIN {X 0,Y 130.249,Z 893.69,A -85,B 0,C 180,E1 -25974.546,E2 -25974.546} C_VEL
LIN {X 0,Y 126.774,Z 901.031,A -85,B 0,C 180,E1 -25977.281,E2 -25977.281} C_VEL
LIN {X 0,Y 122.974,Z 908.483,A -85,B 0,C 180,E1 -25980.936,E2 -25980.936} C_VEL
LIN {X 0,Y 119.01,Z 915.283,A -85,B 0,C 180,E1 -25985.583,E2 -25985.583} C_VEL
LIN {X 0,Y 116.041,Z 920.461,A -85,B 0,C 180,E1 -25990.543,E2 -25990.543} C_VEL
LIN {X 0,Y 113.928,Z 924.267,A -85,B 0,C 180,E1 -25995.715,E2 -25995.715} C_VEL
LIN {X 0,Y 112.97,Z 926.015,A -85,B 0,C 180,E1 -25999.244,E2 -25999.244} C_VEL
LIN {X 0,Y 112.447,Z 927.269,A -85,B 0,C 180,E1 -26002.819,E2 -26002.819} C_VEL
LIN {X 0,Y 112.209,Z 928.048,A -85,B 0,C 180,E1 -26006.409,E2 -26006.409} C_VEL
LIN {X 0,Y 112.262,Z 928.345,A -85,B 0,C 180,E1 -26010,E2 -26010} C_VEL
LIN {X 0,Y 112.206,Z 928.037,A -85,B 0,C 180,E1 -26013.591,E2 -26013.591} C_VEL
LIN {X 0,Y 112.408,Z 927.235,A -85,B 0,C 180,E1 -26017.183,E2 -26017.183} C_VEL
LIN {X 0,Y 112.97,Z 925.959,A -85,B 0,C 180,E1 -26020.756,E2 -26020.756} C_VEL
LIN {X 0,Y 114.512,Z 923.027,A -85,B 0,C 180,E1 -26026.032,E2 -26026.032} C_VEL
LIN {X 0,Y 116.04,Z 920.358,A -85,B 0,C 180,E1 -26029.458,E2 -26029.458} C_VEL
LIN {X 0,Y 119.009,Z 915.15,A -85,B 0,C 180,E1 -26034.417,E2 -26034.417} C_VEL
LIN {X 0,Y 122.966,Z 908.29,A -85,B 0,C 180,E1 -26039.065,E2 -26039.065} C_VEL
LIN {X 0,Y 126.758,Z 900.799,A -85,B 0,C 180,E1 -26042.723,E2 -26042.723} C_VEL
LIN {X 0,Y 130.252,Z 893.416,A -85,B 0,C 180,E1 -26045.453,E2 -26045.453} C_VEL
LIN {X 0,Y 133.406,Z 885.747,A -85,B 0,C 180,E1 -26047.672,E2 -26047.672} C_VEL
LIN {X 0,Y 136.366,Z 877.141,A -85,B 0,C 180,E1 -26049.626,E2 -26049.626} C_VEL
LIN {X 0,Y 139.308,Z 867.008,A -85,B 0,C 180,E1 -26051.329,E2 -26051.329} C_VEL
LIN {X 0,Y 141.74,Z 855.659,A -85,B 0,C 180,E1 -26052.604,E2 -26052.604} C_VEL
LIN {X 0,Y 143.074,Z 846.171,A -85,B 0,C 180,E1 -26053.321,E2 -26053.321} C_VEL
LIN {X 0,Y 144.342,Z 827.097,A -85,B 0,C 180,E1 -26054.266,E2 -26054.266} C_VEL
LIN {X 0,Y 143.857,Z 822.521,A -85,B 0,C 180,E1 -26054.766,E2 -26054.766} C_VEL
LIN {X 0,Y 142.519,Z 818.709,A -85,B 0,C 180,E1 -26055.565,E2 -26055.565} C_VEL
LIN {X 0,Y 140.11,Z 814.388,A -85,B 0,C 180,E1 -26056.886,E2 -26056.886} C_VEL
LIN {X 0,Y 137.247,Z 810.773,A -85,B 0,C 180,E1 -26058.444,E2 -26058.444} C_VEL
LIN {X 0,Y 131.222,Z 804.517,A -85,B 0,C 180,E1 -26062.019,E2 -26062.019} C_VEL
LIN {X 0,Y 127.664,Z 800,A -85,B 0,C 180,E1 -26064.52,E2 -26064.52} C_VEL
LIN {X 0,Y 123.647,Z 794.115,A -85,B 0,C 180,E1 -26067.817,E2 -26067.817} C_VEL
LIN {X 0,Y 120.599,Z 789.872,A -85,B 0,C 180,E1 -26070.672,E2 -26070.672} C_VEL
LIN {X 0,Y 118.083,Z 786.846,A -85,B 0,C 180,E1 -26073.298,E2 -26073.298} C_VEL
LIN {X 0,Y 117.22,Z 785.276,A -85,B 0,C 180,E1 -26074.355,E2 -26074.355} C_VEL
LIN {X 0,Y 114.661,Z 783.046,A -85,B 0,C 180,E1 -26077.482,E2 -26077.482} C_VEL
LIN {X 0,Y 112.81,Z 779.768,A -85,B 0,C 180,E1 -26080.436,E2 -26080.436} C_VEL
LIN {X 0,Y 110.048,Z 777.911,A -85,B 0,C 180,E1 -26085.381,E2 -26085.381} C_VEL
LIN {X 0,Y 108.442,Z 774.593,A -85,B 0,C 180,E1 -26090.676,E2 -26090.676} C_VEL
LIN {X 0,Y 108.371,Z 773.923,A -85,B 0,C 180,E1 -26094.418,E2 -26094.418} C_VEL
LIN {X 0,Y 108.946,Z 773.71,A -85,B 0,C 180,E1 -26100,E2 -26100} C_VEL
LIN {X 0,Y 108.366,Z 774.139,A -85,B 0,C 180,E1 -26107.922,E2 -26107.922} C_VEL
LIN {X 0,Y 108.594,Z 775.046,A -85,B 0,C 180,E1 -26110.724,E2 -26110.724} C_VEL
LIN {X 0,Y 110.227,Z 778.164,A -85,B 0,C 180,E1 -26115.486,E2 -26115.486} C_VEL
LIN {X 0,Y 113.087,Z 780.062,A -85,B 0,C 180,E1 -26120.462,E2 -26120.462} C_VEL
LIN {X 0,Y 114.79,Z 783.237,A -85,B 0,C 180,E1 -26123.16,E2 -26123.16} C_VEL
LIN {X 0,Y 117.471,Z 785.766,A -85,B 0,C 180,E1 -26126.422,E2 -26126.422} C_VEL
LIN {X 0,Y 119.736,Z 789.2,A -85,B 0,C 180,E1 -26128.968,E2 -26128.968} C_VEL
LIN {X 0,Y 121.213,Z 790.692,A -85,B 0,C 180,E1 -26130.389,E2 -26130.389} C_VEL
LIN {X 0,Y 123.892,Z 794.407,A -85,B 0,C 180,E1 -26132.851,E2 -26132.851} C_VEL
LIN {X 0,Y 128.21,Z 800.857,A -85,B 0,C 180,E1 -26136.357,E2 -26136.357} C_VEL
LIN {X 0,Y 133.099,Z 808.778,A -85,B 0,C 180,E1 -26139.81,E2 -26139.81} C_VEL
LIN {X 0,Y 138.02,Z 818.133,A -85,B 0,C 180,E1 -26142.928,E2 -26142.928} C_VEL
LIN {X 0,Y 139.789,Z 821.913,A -85,B 0,C 180,E1 -26143.984,E2 -26143.984} C_VEL
LIN {X 0,Y 138.296,Z 841.643,A -85,B 0,C 180,E1 -26144.968,E2 -26144.968} C_VEL
LIN {X 0,Y 136.282,Z 854.189,A -85,B 0,C 180,E1 -26146.118,E2 -26146.118} C_VEL
LIN {X 0,Y 134.02,Z 863.337,A -85,B 0,C 180,E1 -26147.326,E2 -26147.326} C_VEL
LIN {X 0,Y 131.503,Z 871.943,A -85,B 0,C 180,E1 -26148.917,E2 -26148.917} C_VEL
LIN {X 0,Y 128.875,Z 879.355,A -85,B 0,C 180,E1 -26150.658,E2 -26150.658} C_VEL
LIN {X 0,Y 125.942,Z 886.234,A -85,B 0,C 180,E1 -26152.637,E2 -26152.637} C_VEL
LIN {X 0,Y 122.836,Z 892.917,A -85,B 0,C 180,E1 -26155.1,E2 -26155.1} C_VEL
LIN {X 0,Y 119.419,Z 899.25,A -85,B 0,C 180,E1 -26158.017,E2 -26158.017} C_VEL
LIN {X 0,Y 116.414,Z 904.51,A -85,B 0,C 180,E1 -26161.121,E2 -26161.121} C_VEL
LIN {X 0,Y 113.717,Z 908.9,A -85,B 0,C 180,E1 -26164.366,E2 -26164.366} C_VEL
LIN {X 0,Y 110.373,Z 914.061,A -85,B 0,C 180,E1 -26169.5,E2 -26169.5} C_VEL
LIN {X 0,Y 108.618,Z 916.704,A -85,B 0,C 180,E1 -26173.072,E2 -26173.072} C_VEL
LIN {X 0,Y 106.684,Z 919.597,A -85,B 0,C 180,E1 -26178.602,E2 -26178.602} C_VEL
LIN {X 0,Y 105.833,Z 920.855,A -85,B 0,C 180,E1 -26182.368,E2 -26182.368} C_VEL
LIN {X 0,Y 105.405,Z 921.644,A -85,B 0,C 180,E1 -26186.177,E2 -26186.177} C_VEL
LIN {X 0,Y 105.266,Z 921.944,A -85,B 0,C 180,E1 -26190,E2 -26190} C_VEL
LIN {X 0,Y 105.347,Z 921.664,A -85,B 0,C 180,E1 -26193.825,E2 -26193.825} C_VEL
LIN {X 0,Y 105.832,Z 920.912,A -85,B 0,C 180,E1 -26197.632,E2 -26197.632} C_VEL
LIN {X 0,Y 106.676,Z 919.692,A -85,B 0,C 180,E1 -26201.399,E2 -26201.399} C_VEL
LIN {X 0,Y 108.567,Z 916.839,A -85,B 0,C 180,E1 -26206.936,E2 -26206.936} C_VEL
LIN {X 0,Y 110.315,Z 914.238,A -85,B 0,C 180,E1 -26210.512,E2 -26210.512} C_VEL
LIN {X 0,Y 113.678,Z 909.124,A -85,B 0,C 180,E1 -26215.643,E2 -26215.643} C_VEL
LIN {X 0,Y 117.14,Z 903.617,A -85,B 0,C 180,E1 -26219.668,E2 -26219.668} C_VEL
LIN {X 0,Y 121.027,Z 896.69,A -85,B 0,C 180,E1 -26223.481,E2 -26223.481} C_VEL
LIN {X 0,Y 125.004,Z 888.733,A -85,B 0,C 180,E1 -26226.681,E2 -26226.681} C_VEL
LIN {X 0,Y 128.308,Z 881.145,A -85,B 0,C 180,E1 -26229.043,E2 -26229.043} C_VEL
LIN {X 0,Y 131.211,Z 873.415,A -85,B 0,C 180,E1 -26230.928,E2 -26230.928} C_VEL
LIN {X 0,Y 133.729,Z 865.437,A -85,B 0,C 180,E1 -26232.448,E2 -26232.448} C_VEL
LIN {X 0,Y 136.113,Z 855.867,A -85,B 0,C 180,E1 -26233.829,E2 -26233.829} C_VEL
LIN {X 0,Y 137.731,Z 846.777,A -85,B 0,C 180,E1 -26234.797,E2 -26234.797} C_VEL
LIN {X 0,Y 138.871,Z 837.362,A -85,B 0,C 180,E1 -26235.454,E2 -26235.454} C_VEL
LIN {X 0,Y 139.923,Z 821.957,A -85,B 0,C 180,E1 -26236.193,E2 -26236.193} C_VEL
LIN {X 0,Y 134.931,Z 811.99,A -85,B 0,C 180,E1 -26239.258,E2 -26239.258} C_VEL
LIN {X 0,Y 129.987,Z 803.567,A -85,B 0,C 180,E1 -26242.623,E2 -26242.623} C_VEL
LIN {X 0,Y 126.154,Z 797.73,A -85,B 0,C 180,E1 -26245.556,E2 -26245.556} C_VEL
LIN {X 0,Y 123.744,Z 794.213,A -85,B 0,C 180,E1 -26247.604,E2 -26247.604} C_VEL
LIN {X 0,Y 121.169,Z 790.468,A -85,B 0,C 180,E1 -26250.026,E2 -26250.026} C_VEL
LIN {X 0,Y 118.181,Z 786.928,A -85,B 0,C 180,E1 -26253.128,E2 -26253.128} C_VEL
LIN {X 0,Y 117.172,Z 785.21,A -85,B 0,C 180,E1 -26254.366,E2 -26254.366} C_VEL
LIN {X 0,Y 114.526,Z 782.836,A -85,B 0,C 180,E1 -26257.691,E2 -26257.691} C_VEL
LIN {X 0,Y 112.987,Z 779.937,A -85,B 0,C 180,E1 -26260.231,E2 -26260.231} C_VEL
LIN {X 0,Y 109.939,Z 777.766,A -85,B 0,C 180,E1 -26265.909,E2 -26265.909} C_VEL
LIN {X 0,Y 108.469,Z 774.69,A -85,B 0,C 180,E1 -26271.148,E2 -26271.148} C_VEL
LIN {X 0,Y 108.412,Z 774.009,A -85,B 0,C 180,E1 -26274.419,E2 -26274.419} C_VEL
LIN {X 0,Y 108.946,Z 773.73,A -85,B 0,C 180,E1 -26280,E2 -26280} C_VEL
LIN {X 0,Y 108.427,Z 774.34,A -85,B 0,C 180,E1 -26287.448,E2 -26287.448} C_VEL
LIN {X 0,Y 108.972,Z 776.014,A -85,B 0,C 180,E1 -26290.92,E2 -26290.92} C_VEL
LIN {X 0,Y 111.029,Z 778.817,A -85,B 0,C 180,E1 -26296.077,E2 -26296.077} C_VEL
LIN {X 0,Y 113.186,Z 780.212,A -85,B 0,C 180,E1 -26299.732,E2 -26299.732} C_VEL
LIN {X 0,Y 115.006,Z 783.424,A -85,B 0,C 180,E1 -26302.613,E2 -26302.613} C_VEL
LIN {X 0,Y 117.524,Z 785.716,A -85,B 0,C 180,E1 -26305.693,E2 -26305.693} C_VEL
LIN {X 0,Y 119.746,Z 789.041,A -85,B 0,C 180,E1 -26308.218,E2 -26308.218} C_VEL
LIN {X 0,Y 121.375,Z 790.773,A -85,B 0,C 180,E1 -26309.81,E2 -26309.81} C_VEL
LIN {X 0,Y 124.085,Z 794.537,A -85,B 0,C 180,E1 -26312.311,E2 -26312.311} C_VEL
LIN {X 0,Y 128.261,Z 800.837,A -85,B 0,C 180,E1 -26315.725,E2 -26315.725} C_VEL
LIN {X 0,Y 131.679,Z 806.577,A -85,B 0,C 180,E1 -26318.227,E2 -26318.227} C_VEL
LIN {X 0,Y 135.841,Z 816.182,A -85,B 0,C 180,E1 -26321.149,E2 -26321.149} C_VEL
LIN {X 0,Y 139.288,Z 826.103,A -85,B 0,C 180,E1 -26323.467,E2 -26323.467} C_VEL
LIN {X 0,Y 139.403,Z 830.562,A -85,B 0,C 180,E1 -26323.841,E2 -26323.841} C_VEL
LIN {X 0,Y 137.941,Z 848.13,A -85,B 0,C 180,E1 -26324.705,E2 -26324.705} C_VEL
LIN {X 0,Y 136.06,Z 859.149,A -85,B 0,C 180,E1 -26325.669,E2 -26325.669} C_VEL
LIN {X 0,Y 133.657,Z 868.684,A -85,B 0,C 180,E1 -26326.877,E2 -26326.877} C_VEL
LIN {X 0,Y 131.001,Z 877.351,A -85,B 0,C 180,E1 -26328.402,E2 -26328.402} C_VEL
LIN {X 0,Y 128.261,Z 884.823,A -85,B 0,C 180,E1 -26330.095,E2 -26330.095} C_VEL
LIN {X 0,Y 125.008,Z 892.461,A -85,B 0,C 180,E1 -26332.309,E2 -26332.309} C_VEL
LIN {X 0,Y 121.767,Z 899.117,A -85,B 0,C 180,E1 -26334.748,E2 -26334.748} C_VEL
LIN {X 0,Y 118.356,Z 905.439,A -85,B 0,C 180,E1 -26337.695,E2 -26337.695} C_VEL
LIN {X 0,Y 115.302,Z 910.693,A -85,B 0,C 180,E1 -26340.816,E2 -26340.816} C_VEL
LIN {X 0,Y 112.58,Z 915.075,A -85,B 0,C 180,E1 -26344.088,E2 -26344.088} C_VEL
LIN {X 0,Y 109.337,Z 920.253,A -85,B 0,C 180,E1 -26349.297,E2 -26349.297} C_VEL
LIN {X 0,Y 107.031,Z 924.058,A -85,B 0,C 180,E1 -26354.772,E2 -26354.772} C_VEL
LIN {X 0,Y 105.999,Z 925.806,A -85,B 0,C 180,E1 -26358.527,E2 -26358.527} C_VEL
LIN {X 0,Y 105.384,Z 927.06,A -85,B 0,C 180,E1 -26362.335,E2 -26362.335} C_VEL
LIN {X 0,Y 105.121,Z 927.839,A -85,B 0,C 180,E1 -26366.167,E2 -26366.167} C_VEL
LIN {X 0,Y 105.175,Z 928.137,A -85,B 0,C 180,E1 -26370,E2 -26370} C_VEL
LIN {X 0,Y 105.117,Z 927.828,A -85,B 0,C 180,E1 -26373.834,E2 -26373.834} C_VEL
LIN {X 0,Y 105.349,Z 927.025,A -85,B 0,C 180,E1 -26377.667,E2 -26377.667} C_VEL
LIN {X 0,Y 105.998,Z 925.749,A -85,B 0,C 180,E1 -26381.473,E2 -26381.473} C_VEL
LIN {X 0,Y 107.696,Z 922.817,A -85,B 0,C 180,E1 -26387.077,E2 -26387.077} C_VEL
LIN {X 0,Y 109.336,Z 920.147,A -85,B 0,C 180,E1 -26390.704,E2 -26390.704} C_VEL
LIN {X 0,Y 112.579,Z 914.939,A -85,B 0,C 180,E1 -26395.912,E2 -26395.912} C_VEL
LIN {X 0,Y 116.815,Z 908.079,A -85,B 0,C 180,E1 -26400.756,E2 -26400.756} C_VEL
LIN {X 0,Y 120.85,Z 900.588,A -85,B 0,C 180,E1 -26404.542,E2 -26404.542} C_VEL
LIN {X 0,Y 124.535,Z 893.204,A -85,B 0,C 180,E1 -26407.349,E2 -26407.349} C_VEL
LIN {X 0,Y 127.753,Z 885.801,A -85,B 0,C 180,E1 -26409.546,E2 -26409.546} C_VEL
LIN {X 0,Y 130.97,Z 876.927,A -85,B 0,C 180,E1 -26411.61,E2 -26411.61} C_VEL
LIN {X 0,Y 134.024,Z 866.885,A -85,B 0,C 180,E1 -26413.323,E2 -26413.323} C_VEL
LIN {X 0,Y 136.583,Z 855.487,A -85,B 0,C 180,E1 -26414.619,E2 -26414.619} C_VEL
LIN {X 0,Y 137.997,Z 845.946,A -85,B 0,C 180,E1 -26415.344,E2 -26415.344} C_VEL
LIN {X 0,Y 139.257,Z 828.258,A -85,B 0,C 180,E1 -26416.24,E2 -26416.24} C_VEL
LIN {X 0,Y 138.809,Z 824.846,A -85,B 0,C 180,E1 -26416.683,E2 -26416.683} C_VEL
LIN {X 0,Y 134.952,Z 814.15,A -85,B 0,C 180,E1 -26419.277,E2 -26419.277} C_VEL
LIN {X 0,Y 130.771,Z 804.93,A -85,B 0,C 180,E1 -26422.234,E2 -26422.234} C_VEL
LIN {X 0,Y 127.664,Z 800,A -85,B 0,C 180,E1 -26424.52,E2 -26424.52} C_VEL
LIN {X 0,Y 125.85,Z 798.189,A -85,B 0,C 180,E1 -26425.864,E2 -26425.864} C_VEL
LIN {X 0,Y 122.38,Z 797.056,A -85,B 0,C 180,E1 -26428.441,E2 -26428.441} C_VEL
LIN {X 0,Y 118.41,Z 796.025,A -85,B 0,C 180,E1 -26431.82,E2 -26431.82} C_VEL
LIN {X 0,Y 117.323,Z 795.098,A -85,B 0,C 180,E1 -26432.938,E2 -26432.938} C_VEL
LIN {X 0,Y 115.098,Z 791.686,A -85,B 0,C 180,E1 -26435.667,E2 -26435.667} C_VEL
LIN {X 0,Y 112.595,Z 789.11,A -85,B 0,C 180,E1 -26439.063,E2 -26439.063} C_VEL
LIN {X 0,Y 111.327,Z 786.594,A -85,B 0,C 180,E1 -26441.302,E2 -26441.302} C_VEL
LIN {X 0,Y 108.73,Z 784.648,A -85,B 0,C 180,E1 -26446.33,E2 -26446.33} C_VEL
LIN {X 0,Y 107.181,Z 781.408,A -85,B 0,C 180,E1 -26451.516,E2 -26451.516} C_VEL
LIN {X 0,Y 106.307,Z 780.584,A -85,B 0,C 180,E1 -26456.21,E2 -26456.21} C_VEL
LIN {X 0,Y 106.091,Z 780.221,A -85,B 0,C 180,E1 -26460,E2 -26460} C_VEL
LIN {X 0,Y 107.069,Z 781.299,A -85,B 0,C 180,E1 -26468.493,E2 -26468.493} C_VEL
LIN {X 0,Y 107.57,Z 782.445,A -85,B 0,C 180,E1 -26470.589,E2 -26470.589} C_VEL
LIN {X 0,Y 109.065,Z 785.096,A -85,B 0,C 180,E1 -26474.937,E2 -26474.937} C_VEL
LIN {X 0,Y 111.481,Z 786.915,A -85,B 0,C 180,E1 -26479.448,E2 -26479.448} C_VEL
LIN {X 0,Y 113.42,Z 790.281,A -85,B 0,C 180,E1 -26482.639,E2 -26482.639} C_VEL
LIN {X 0,Y 115.424,Z 792.269,A -85,B 0,C 180,E1 -26485.228,E2 -26485.228} C_VEL
LIN {X 0,Y 117.777,Z 795.748,A -85,B 0,C 180,E1 -26488.029,E2 -26488.029} C_VEL
LIN {X 0,Y 118.978,Z 797.182,A -85,B 0,C 180,E1 -26489.283,E2 -26489.283} C_VEL
LIN {X 0,Y 122.175,Z 801.907,A -85,B 0,C 180,E1 -26492.391,E2 -26492.391} C_VEL
LIN {X 0,Y 126.068,Z 807.854,A -85,B 0,C 180,E1 -26495.68,E2 -26495.68} C_VEL
LIN {X 0,Y 131.471,Z 817.523,A -85,B 0,C 180,E1 -26499.686,E2 -26499.686} C_VEL
LIN {X 0,Y 134.79,Z 824.473,A -85,B 0,C 180,E1 -26501.919,E2 -26501.919} C_VEL
LIN {X 0,Y 133.381,Z 841.868,A -85,B 0,C 180,E1 -26502.814,E2 -26502.814} C_VEL
LIN {X 0,Y 131.346,Z 854.046,A -85,B 0,C 180,E1 -26503.928,E2 -26503.928} C_VEL
LIN {X 0,Y 128.91,Z 863.551,A -85,B 0,C 180,E1 -26505.195,E2 -26505.195} C_VEL
LIN {X 0,Y 126.11,Z 872.548,A -85,B 0,C 180,E1 -26506.887,E2 -26506.887} C_VEL
LIN {X 0,Y 123.481,Z 879.567,A -85,B 0,C 180,E1 -26508.575,E2 -26508.575} C_VEL
LIN {X 0,Y 120.391,Z 886.446,A -85,B 0,C 180,E1 -26510.592,E2 -26510.592} C_VEL
LIN {X 0,Y 117.102,Z 893.128,A -85,B 0,C 180,E1 -26513.119,E2 -26513.119} C_VEL
LIN {X 0,Y 113.474,Z 899.461,A -85,B 0,C 180,E1 -26516.123,E2 -26516.123} C_VEL
LIN {X 0,Y 110.25,Z 904.721,A -85,B 0,C 180,E1 -26519.338,E2 -26519.338} C_VEL
LIN {X 0,Y 107.372,Z 909.11,A -85,B 0,C 180,E1 -26522.73,E2 -26522.73} C_VEL
LIN {X 0,Y 103.764,Z 914.271,A -85,B 0,C 180,E1 -26528.129,E2 -26528.129} C_VEL
LIN {X 0,Y 101.856,Z 916.913,A -85,B 0,C 180,E1 -26531.911,E2 -26531.911} C_VEL
LIN {X 0,Y 99.75,Z 919.806,A -85,B 0,C 180,E1 -26537.797,E2 -26537.797} C_VEL
LIN {X 0,Y 98.822,Z 921.064,A -85,B 0,C 180,E1 -26541.823,E2 -26541.823} C_VEL
LIN {X 0,Y 98.33,Z 921.853,A -85,B 0,C 180,E1 -26545.901,E2 -26545.901} C_VEL
LIN {X 0,Y 98.192,Z 922.152,A -85,B 0,C 180,E1 -26550,E2 -26550} C_VEL
LIN {X 0,Y 98.281,Z 921.873,A -85,B 0,C 180,E1 -26554.101,E2 -26554.101} C_VEL
LIN {X 0,Y 98.821,Z 921.12,A -85,B 0,C 180,E1 -26558.177,E2 -26558.177} C_VEL
LIN {X 0,Y 99.741,Z 919.899,A -85,B 0,C 180,E1 -26562.204,E2 -26562.204} C_VEL
LIN {X 0,Y 101.811,Z 917.046,A -85,B 0,C 180,E1 -26568.097,E2 -26568.097} C_VEL
LIN {X 0,Y 103.693,Z 914.446,A -85,B 0,C 180,E1 -26571.887,E2 -26571.887} C_VEL
LIN {X 0,Y 107.336,Z 909.331,A -85,B 0,C 180,E1 -26577.28,E2 -26577.28} C_VEL
LIN {X 0,Y 111.037,Z 903.824,A -85,B 0,C 180,E1 -26581.478,E2 -26581.478} C_VEL
LIN {X 0,Y 115.169,Z 896.897,A -85,B 0,C 180,E1 -26585.431,E2 -26585.431} C_VEL
LIN {X 0,Y 119.387,Z 888.939,A -85,B 0,C 180,E1 -26588.716,E2 -26588.716} C_VEL
LIN {X 0,Y 122.886,Z 881.35,A -85,B 0,C 180,E1 -26591.124,E2 -26591.124} C_VEL
LIN {X 0,Y 125.857,Z 873.86,A -85,B 0,C 180,E1 -26592.989,E2 -26592.989} C_VEL
LIN {X 0,Y 128.58,Z 865.639,A -85,B 0,C 180,E1 -26594.583,E2 -26594.583} C_VEL
LIN {X 0,Y 130.861,Z 857.078,A -85,B 0,C 180,E1 -26595.848,E2 -26595.848} C_VEL
LIN {X 0,Y 132.592,Z 848.241,A -85,B 0,C 180,E1 -26596.834,E2 -26596.834} C_VEL
LIN {X 0,Y 133.748,Z 839.905,A -85,B 0,C 180,E1 -26597.478,E2 -26597.478} C_VEL
LIN {X 0,Y 134.887,Z 824.469,A -85,B 0,C 180,E1 -26598.289,E2 -26598.289} C_VEL
LIN {X 0,Y 130.845,Z 816.192,A -85,B 0,C 180,E1 -26601.034,E2 -26601.034} C_VEL
LIN {X 0,Y 125.974,Z 807.587,A -85,B 0,C 180,E1 -26604.708,E2 -26604.708} C_VEL
LIN {X 0,Y 121.275,Z 800.361,A -85,B 0,C 180,E1 -26608.806,E2 -26608.806} C_VEL
LIN {X 0,Y 118.274,Z 796.063,A -85,B 0,C 180,E1 -26611.858,E2 -26611.858} C_VEL
LIN {X 0,Y 115.714,Z 792.621,A -85,B 0,C 180,E1 -26614.839,E2 -26614.839} C_VEL
LIN {X 0,Y 115.084,Z 791.652,A -85,B 0,C 180,E1 -26615.665,E2 -26615.665} C_VEL
LIN {X 0,Y 112.63,Z 789.121,A -85,B 0,C 180,E1 -26619.063,E2 -26619.063} C_VEL
LIN {X 0,Y 111.223,Z 786.551,A -85,B 0,C 180,E1 -26621.582,E2 -26621.582} C_VEL
LIN {X 0,Y 108.589,Z 784.414,A -85,B 0,C 180,E1 -26627.04,E2 -26627.04} C_VEL
LIN {X 0,Y 107.254,Z 781.513,A -85,B 0,C 180,E1 -26631.995,E2 -26631.995} C_VEL
LIN {X 0,Y 106.424,Z 780.537,A -85,B 0,C 180,E1 -26638.107,E2 -26638.107} C_VEL
LIN {X 0,Y 106.447,Z 780.533,A -85,B 0,C 180,E1 -26641.891,E2 -26641.891} C_VEL
LIN {X 0,Y 107.281,Z 781.56,A -85,B 0,C 180,E1 -26647.765,E2 -26647.765} C_VEL
LIN {X 0,Y 109.687,Z 785.607,A -85,B 0,C 180,E1 -26655.206,E2 -26655.206} C_VEL
LIN {X 0,Y 111.519,Z 786.9,A -85,B 0,C 180,E1 -26658.575,E2 -26658.575} C_VEL
LIN {X 0,Y 113.597,Z 790.377,A -85,B 0,C 180,E1 -26662.027,E2 -26662.027} C_VEL
LIN {X 0,Y 115.51,Z 792.226,A -85,B 0,C 180,E1 -26664.516,E2 -26664.516} C_VEL
LIN {X 0,Y 118,Z 795.803,A -85,B 0,C 180,E1 -26667.489,E2 -26667.489} C_VEL
LIN {X 0,Y 119.039,Z 797.089,A -85,B 0,C 180,E1 -26668.586,E2 -26668.586} C_VEL
LIN {X 0,Y 122.406,Z 802.114,A -85,B 0,C 180,E1 -26671.886,E2 -26671.886} C_VEL
LIN {X 0,Y 125.427,Z 806.787,A -85,B 0,C 180,E1 -26674.488,E2 -26674.488} C_VEL
LIN {X 0,Y 128.332,Z 811.983,A -85,B 0,C 180,E1 -26676.797,E2 -26676.797} C_VEL
LIN {X 0,Y 132.075,Z 821.302,A -85,B 0,C 180,E1 -26679.683,E2 -26679.683} C_VEL
LIN {X 0,Y 134.523,Z 828.572,A -85,B 0,C 180,E1 -26681.491,E2 -26681.491} C_VEL
LIN {X 0,Y 134.092,Z 837.188,A -85,B 0,C 180,E1 -26681.962,E2 -26681.962} C_VEL
LIN {X 0,Y 132.619,Z 850.735,A -85,B 0,C 180,E1 -26682.75,E2 -26682.75} C_VEL
LIN {X 0,Y 130.913,Z 859.615,A -85,B 0,C 180,E1 -26683.579,E2 -26683.579} C_VEL
LIN {X 0,Y 128.578,Z 868.482,A -85,B 0,C 180,E1 -26684.719,E2 -26684.719} C_VEL
LIN {X 0,Y 125.777,Z 877.146,A -85,B 0,C 180,E1 -26686.253,E2 -26686.253} C_VEL
LIN {X 0,Y 122.753,Z 884.946,A -85,B 0,C 180,E1 -26688.057,E2 -26688.057} C_VEL
LIN {X 0,Y 119.468,Z 892.256,A -85,B 0,C 180,E1 -26690.227,E2 -26690.227} C_VEL
LIN {X 0,Y 116.052,Z 898.911,A -85,B 0,C 180,E1 -26692.728,E2 -26692.728} C_VEL
LIN {X 0,Y 112.403,Z 905.231,A -85,B 0,C 180,E1 -26695.756,E2 -26695.756} C_VEL
LIN {X 0,Y 109.162,Z 910.486,A -85,B 0,C 180,E1 -26698.999,E2 -26698.999} C_VEL
LIN {X 0,Y 106.241,Z 914.868,A -85,B 0,C 180,E1 -26702.415,E2 -26702.415} C_VEL
LIN {X 0,Y 102.701,Z 920.044,A -85,B 0,C 180,E1 -26707.891,E2 -26707.891} C_VEL
LIN {X 0,Y 100.181,Z 923.849,A -85,B 0,C 180,E1 -26713.703,E2 -26713.703} C_VEL
LIN {X 0,Y 99.031,Z 925.597,A -85,B 0,C 180,E1 -26717.707,E2 -26717.707} C_VEL
LIN {X 0,Y 98.339,Z 926.851,A -85,B 0,C 180,E1 -26721.782,E2 -26721.782} C_VEL
LIN {X 0,Y 98.033,Z 927.63,A -85,B 0,C 180,E1 -26725.889,E2 -26725.889} C_VEL
LIN {X 0,Y 98.08,Z 927.928,A -85,B 0,C 180,E1 -26730,E2 -26730} C_VEL
LIN {X 0,Y 98.029,Z 927.619,A -85,B 0,C 180,E1 -26734.111,E2 -26734.111} C_VEL
LIN {X 0,Y 98.312,Z 926.815,A -85,B 0,C 180,E1 -26738.22,E2 -26738.22} C_VEL
LIN {X 0,Y 99.031,Z 925.539,A -85,B 0,C 180,E1 -26742.293,E2 -26742.293} C_VEL
LIN {X 0,Y 100.928,Z 922.607,A -85,B 0,C 180,E1 -26748.261,E2 -26748.261} C_VEL
LIN {X 0,Y 102.7,Z 919.936,A -85,B 0,C 180,E1 -26752.11,E2 -26752.11} C_VEL
LIN {X 0,Y 106.24,Z 914.729,A -85,B 0,C 180,E1 -26757.585,E2 -26757.585} C_VEL
LIN {X 0,Y 110.772,Z 907.868,A -85,B 0,C 180,E1 -26762.635,E2 -26762.635} C_VEL
LIN {X 0,Y 115.08,Z 900.376,A -85,B 0,C 180,E1 -26766.544,E2 -26766.544} C_VEL
LIN {X 0,Y 118.971,Z 892.992,A -85,B 0,C 180,E1 -26769.423,E2 -26769.423} C_VEL
LIN {X 0,Y 122.32,Z 885.667,A -85,B 0,C 180,E1 -26771.645,E2 -26771.645} C_VEL
LIN {X 0,Y 125.213,Z 878.217,A -85,B 0,C 180,E1 -26773.438,E2 -26773.438} C_VEL
LIN {X 0,Y 127.971,Z 869.817,A -85,B 0,C 180,E1 -26774.998,E2 -26774.998} C_VEL
LIN {X 0,Y 130.423,Z 860.902,A -85,B 0,C 180,E1 -26776.189,E2 -26776.189} C_VEL
LIN {X 0,Y 132.556,Z 850.11,A -85,B 0,C 180,E1 -26777.223,E2 -26777.223} C_VEL
LIN {X 0,Y 134.059,Z 835.11,A -85,B 0,C 180,E1 -26778.054,E2 -26778.054} C_VEL
LIN {X 0,Y 134.325,Z 828.585,A -85,B 0,C 180,E1 -26778.439,E2 -26778.439} C_VEL
LIN {X 0,Y 131.694,Z 820.537,A -85,B 0,C 180,E1 -26780.403,E2 -26780.403} C_VEL
LIN {X 0,Y 127.921,Z 811.312,A -85,B 0,C 180,E1 -26783.311,E2 -26783.311} C_VEL
LIN {X 0,Y 124.862,Z 806.009,A -85,B 0,C 180,E1 -26785.747,E2 -26785.747} C_VEL
LIN {X 0,Y 121.168,Z 800.252,A -85,B 0,C 180,E1 -26789.018,E2 -26789.018} C_VEL
LIN {X 0,Y 118.176,Z 796.01,A -85,B 0,C 180,E1 -26792.032,E2 -26792.032} C_VEL
LIN {X 0,Y 117.323,Z 795.098,A -85,B 0,C 180,E1 -26792.938,E2 -26792.938} C_VEL
LIN {X 0,Y 115.783,Z 793.891,A -85,B 0,C 180,E1 -26794.623,E2 -26794.623} C_VEL
LIN {X 0,Y 113.13,Z 793.437,A -85,B 0,C 180,E1 -26797.662,E2 -26797.662} C_VEL
LIN {X 0,Y 110.255,Z 793.488,A -85,B 0,C 180,E1 -26801.572,E2 -26801.572} C_VEL
LIN {X 0,Y 109.46,Z 793.184,A -85,B 0,C 180,E1 -26802.912,E2 -26802.912} C_VEL
LIN {X 0,Y 107.203,Z 791,A -85,B 0,C 180,E1 -26807.99,E2 -26807.99} C_VEL
LIN {X 0,Y 106.096,Z 788.252,A -85,B 0,C 180,E1 -26812.387,E2 -26812.387} C_VEL
LIN {X 0,Y 105.224,Z 787.277,A -85,B 0,C 180,E1 -26820,E2 -26820} C_VEL
LIN {X 0,Y 106.097,Z 788.291,A -85,B 0,C 180,E1 -26828.092,E2 -26828.092} C_VEL
LIN {X 0,Y 107.819,Z 791.9,A -85,B 0,C 180,E1 -26834.142,E2 -26834.142} C_VEL
LIN {X 0,Y 109.861,Z 793.609,A -85,B 0,C 180,E1 -26838.293,E2 -26838.293} C_VEL
LIN {X 0,Y 111.921,Z 797.098,A -85,B 0,C 180,E1 -26841.89,E2 -26841.89} C_VEL
LIN {X 0,Y 113.476,Z 798.816,A -85,B 0,C 180,E1 -26844.053,E2 -26844.053} C_VEL
LIN {X 0,Y 116.079,Z 802.522,A -85,B 0,C 180,E1 -26847.311,E2 -26847.311} C_VEL
LIN {X 0,Y 119.42,Z 807.619,A -85,B 0,C 180,E1 -26850.89,E2 -26850.89} C_VEL
LIN {X 0,Y 122.965,Z 813.32,A -85,B 0,C 180,E1 -26854.16,E2 -26854.16} C_VEL
LIN {X 0,Y 128.016,Z 822.815,A -85,B 0,C 180,E1 -26858.243,E2 -26858.243} C_VEL
LIN {X 0,Y 130.011,Z 827.19,A -85,B 0,C 180,E1 -26859.728,E2 -26859.728} C_VEL
LIN {X 0,Y 128.56,Z 843.134,A -85,B 0,C 180,E1 -26860.566,E2 -26860.566} C_VEL
LIN {X 0,Y 126.546,Z 854.231,A -85,B 0,C 180,E1 -26861.615,E2 -26861.615} C_VEL
LIN {X 0,Y 124.366,Z 862.653,A -85,B 0,C 180,E1 -26862.723,E2 -26862.723} C_VEL
LIN {X 0,Y 121.76,Z 870.742,A -85,B 0,C 180,E1 -26864.144,E2 -26864.144} C_VEL
LIN {X 0,Y 118.267,Z 879.779,A -85,B 0,C 180,E1 -26866.305,E2 -26866.305} C_VEL
LIN {X 0,Y 114.499,Z 887.676,A -85,B 0,C 180,E1 -26868.712,E2 -26868.712} C_VEL
LIN {X 0,Y 110.521,Z 895.037,A -85,B 0,C 180,E1 -26871.684,E2 -26871.684} C_VEL
LIN {X 0,Y 105.909,Z 902.494,A -85,B 0,C 180,E1 -26875.664,E2 -26875.664} C_VEL
LIN {X 0,Y 101.128,Z 909.32,A -85,B 0,C 180,E1 -26880.891,E2 -26880.891} C_VEL
LIN {X 0,Y 97.227,Z 914.48,A -85,B 0,C 180,E1 -26886.574,E2 -26886.574} C_VEL
LIN {X 0,Y 95.125,Z 917.123,A -85,B 0,C 180,E1 -26890.581,E2 -26890.581} C_VEL
LIN {X 0,Y 92.817,Z 920.016,A -85,B 0,C 180,E1 -26896.87,E2 -26896.87} C_VEL
LIN {X 0,Y 91.811,Z 921.273,A -85,B 0,C 180,E1 -26901.194,E2 -26901.194} C_VEL
LIN {X 0,Y 91.25,Z 922.062,A -85,B 0,C 180,E1 -26905.583,E2 -26905.583} C_VEL
LIN {X 0,Y 91.115,Z 922.361,A -85,B 0,C 180,E1 -26910,E2 -26910} C_VEL
LIN {X 0,Y 91.22,Z 922.081,A -85,B 0,C 180,E1 -26914.419,E2 -26914.419} C_VEL
LIN {X 0,Y 91.811,Z 921.328,A -85,B 0,C 180,E1 -26918.807,E2 -26918.807} C_VEL
LIN {X 0,Y 92.805,Z 920.108,A -85,B 0,C 180,E1 -26923.131,E2 -26923.131} C_VEL
LIN {X 0,Y 95.081,Z 917.255,A -85,B 0,C 180,E1 -26929.428,E2 -26929.428} C_VEL
LIN {X 0,Y 97.133,Z 914.654,A -85,B 0,C 180,E1 -26933.45,E2 -26933.45} C_VEL
LIN {X 0,Y 101.096,Z 909.538,A -85,B 0,C 180,E1 -26939.119,E2 -26939.119} C_VEL
LIN {X 0,Y 105.038,Z 904.031,A -85,B 0,C 180,E1 -26943.504,E2 -26943.504} C_VEL
LIN {X 0,Y 109.467,Z 897.103,A -85,B 0,C 180,E1 -26947.584,E2 -26947.584} C_VEL
LIN {X 0,Y 113.935,Z 889.144,A -85,B 0,C 180,E1 -26950.95,E2 -26950.95} C_VEL
LIN {X 0,Y 117.645,Z 881.554,A -85,B 0,C 180,E1 -26953.393,E2 -26953.393} C_VEL
LIN {X 0,Y 121.101,Z 873.158,A -85,B 0,C 180,E1 -26955.481,E2 -26955.481} C_VEL
LIN {X 0,Y 123.997,Z 864.668,A -85,B 0,C 180,E1 -26957.083,E2 -26957.083} C_VEL
LIN {X 0,Y 126.295,Z 856.086,A -85,B 0,C 180,E1 -26958.32,E2 -26958.32} C_VEL
LIN {X 0,Y 128.175,Z 846.448,A -85,B 0,C 180,E1 -26959.343,E2 -26959.343} C_VEL
LIN {X 0,Y 129.567,Z 835.45,A -85,B 0,C 180,E1 -26960.071,E2 -26960.071} C_VEL
LIN {X 0,Y 130.144,Z 827.225,A -85,B 0,C 180,E1 -26960.469,E2 -26960.469} C_VEL
LIN {X 0,Y 126.055,Z 818.791,A -85,B 0,C 180,E1 -26963.583,E2 -26963.583} C_VEL
LIN {X 0,Y 121.086,Z 809.999,A -85,B 0,C 180,E1 -26967.88,E2 -26967.88} C_VEL
LIN {X 0,Y 117.908,Z 805.258,A -85,B 0,C 180,E1 -26971.033,E2 -26971.033} C_VEL
LIN {X 0,Y 115.763,Z 801.992,A -85,B 0,C 180,E1 -26973.473,E2 -26973.473} C_VEL
LIN {X 0,Y 113.041,Z 798.053,A -85,B 0,C 180,E1 -26977.038,E2 -26977.038} C_VEL
LIN {X 0,Y 110.54,Z 794.942,A -85,B 0,C 180,E1 -26980.959,E2 -26980.959} C_VEL
LIN {X 0,Y 109.82,Z 793.38,A -85,B 0,C 180,E1 -26982.423,E2 -26982.423} C_VEL
LIN {X 0,Y 107.323,Z 791.128,A -85,B 0,C 180,E1 -26988.07,E2 -26988.07} C_VEL
LIN {X 0,Y 106.194,Z 788.363,A -85,B 0,C 180,E1 -26992.871,E2 -26992.871} C_VEL
LIN {X 0,Y 105.532,Z 787.421,A -85,B 0,C 180,E1 -27000,E2 -27000} C_VEL
LIN {X 0,Y 106.237,Z 788.428,A -85,B 0,C 180,E1 -27006.98,E2 -27006.98} C_VEL
LIN {X 0,Y 108.367,Z 792.371,A -85,B 0,C 180,E1 -27014.299,E2 -27014.299} C_VEL
LIN {X 0,Y 109.989,Z 793.671,A -85,B 0,C 180,E1 -27017.548,E2 -27017.548} C_VEL
LIN {X 0,Y 111.949,Z 797.004,A -85,B 0,C 180,E1 -27021.041,E2 -27021.041} C_VEL
LIN {X 0,Y 113.589,Z 798.751,A -85,B 0,C 180,E1 -27023.351,E2 -27023.351} C_VEL
LIN {X 0,Y 116.212,Z 802.492,A -85,B 0,C 180,E1 -27026.669,E2 -27026.669} C_VEL
LIN {X 0,Y 120.178,Z 808.667,A -85,B 0,C 180,E1 -27030.899,E2 -27030.899} C_VEL
LIN {X 0,Y 124.257,Z 815.568,A -85,B 0,C 180,E1 -27034.582,E2 -27034.582} C_VEL
LIN {X 0,Y 127.664,Z 824.25,A -85,B 0,C 180,E1 -27037.517,E2 -27037.517} C_VEL
LIN {X 0,Y 129.854,Z 830.976,A -85,B 0,C 180,E1 -27039.326,E2 -27039.326} C_VEL
LIN {X 0,Y 128.306,Z 848.174,A -85,B 0,C 180,E1 -27040.229,E2 -27040.229} C_VEL
LIN {X 0,Y 125.943,Z 860.106,A -85,B 0,C 180,E1 -27041.321,E2 -27041.321} C_VEL
LIN {X 0,Y 123.681,Z 868.279,A -85,B 0,C 180,E1 -27042.379,E2 -27042.379} C_VEL
LIN {X 0,Y 120.752,Z 876.942,A -85,B 0,C 180,E1 -27043.925,E2 -27043.925} C_VEL
LIN {X 0,Y 117.301,Z 885.34,A -85,B 0,C 180,E1 -27045.909,E2 -27045.909} C_VEL
LIN {X 0,Y 113.574,Z 893.073,A -85,B 0,C 180,E1 -27048.301,E2 -27048.301} C_VEL
LIN {X 0,Y 109.477,Z 900.413,A -85,B 0,C 180,E1 -27051.251,E2 -27051.251} C_VEL
LIN {X 0,Y 104.872,Z 907.863,A -85,B 0,C 180,E1 -27055.276,E2 -27055.276} C_VEL
LIN {X 0,Y 100.758,Z 913.701,A -85,B 0,C 180,E1 -27059.622,E2 -27059.622} C_VEL
LIN {X 0,Y 97.267,Z 918.308,A -85,B 0,C 180,E1 -27064.308,E2 -27064.308} C_VEL
LIN {X 0,Y 95.122,Z 921.309,A -85,B 0,C 180,E1 -27068.32,E2 -27068.32} C_VEL
LIN {X 0,Y 93.382,Z 923.641,A -85,B 0,C 180,E1 -27072.48,E2 -27072.48} C_VEL
LIN {X 0,Y 92.098,Z 925.389,A -85,B 0,C 180,E1 -27076.766,E2 -27076.766} C_VEL
LIN {X 0,Y 91.318,Z 926.642,A -85,B 0,C 180,E1 -27081.146,E2 -27081.146} C_VEL
LIN {X 0,Y 90.943,Z 927.421,A -85,B 0,C 180,E1 -27085.568,E2 -27085.568} C_VEL
LIN {X 0,Y 90.978,Z 927.719,A -85,B 0,C 180,E1 -27090,E2 -27090} C_VEL
LIN {X 0,Y 90.938,Z 927.409,A -85,B 0,C 180,E1 -27094.432,E2 -27094.432} C_VEL
LIN {X 0,Y 91.298,Z 926.606,A -85,B 0,C 180,E1 -27098.856,E2 -27098.856} C_VEL
LIN {X 0,Y 92.098,Z 925.329,A -85,B 0,C 180,E1 -27103.234,E2 -27103.234} C_VEL
LIN {X 0,Y 94.194,Z 922.397,A -85,B 0,C 180,E1 -27109.618,E2 -27109.618} C_VEL
LIN {X 0,Y 96.141,Z 919.725,A -85,B 0,C 180,E1 -27113.707,E2 -27113.707} C_VEL
LIN {X 0,Y 100.008,Z 914.519,A -85,B 0,C 180,E1 -27119.467,E2 -27119.467} C_VEL
LIN {X 0,Y 104.845,Z 907.657,A -85,B 0,C 180,E1 -27124.734,E2 -27124.734} C_VEL
LIN {X 0,Y 109.468,Z 900.165,A -85,B 0,C 180,E1 -27128.753,E2 -27128.753} C_VEL
LIN {X 0,Y 113.569,Z 892.78,A -85,B 0,C 180,E1 -27131.701,E2 -27131.701} C_VEL
LIN {X 0,Y 116.946,Z 885.827,A -85,B 0,C 180,E1 -27133.851,E2 -27133.851} C_VEL
LIN {X 0,Y 120.156,Z 878.003,A -85,B 0,C 180,E1 -27135.767,E2 -27135.767} C_VEL
LIN {X 0,Y 123.068,Z 869.603,A -85,B 0,C 180,E1 -27137.328,E2 -27137.328} C_VEL
LIN {X 0,Y 125.474,Z 861.281,A -85,B 0,C 180,E1 -27138.45,E2 -27138.45} C_VEL
LIN {X 0,Y 127.55,Z 851.405,A -85,B 0,C 180,E1 -27139.435,E2 -27139.435} C_VEL
LIN {X 0,Y 129.064,Z 839.577,A -85,B 0,C 180,E1 -27140.183,E2 -27140.183} C_VEL
LIN {X 0,Y 129.655,Z 830.725,A -85,B 0,C 180,E1 -27140.621,E2 -27140.621} C_VEL
LIN {X 0,Y 126.109,Z 820.348,A -85,B 0,C 180,E1 -27143.569,E2 -27143.569} C_VEL
LIN {X 0,Y 123.48,Z 814.334,A -85,B 0,C 180,E1 -27145.843,E2 -27145.843} C_VEL
LIN {X 0,Y 120.158,Z 808.766,A -85,B 0,C 180,E1 -27148.851,E2 -27148.851} C_VEL
LIN {X 0,Y 117.912,Z 805.306,A -85,B 0,C 180,E1 -27151.111,E2 -27151.111} C_VEL
LIN {X 0,Y 115.722,Z 801.995,A -85,B 0,C 180,E1 -27153.567,E2 -27153.567} C_VEL
LIN {X 0,Y 112.955,Z 798.031,A -85,B 0,C 180,E1 -27157.136,E2 -27157.136} C_VEL
LIN {X 0,Y 110.53,Z 795.01,A -85,B 0,C 180,E1 -27160.861,E2 -27160.861} C_VEL
LIN {X 0,Y 109.801,Z 793.427,A -85,B 0,C 180,E1 -27162.3,E2 -27162.3} C_VEL
LIN {X 0,Y 109.46,Z 793.184,A -85,B 0,C 180,E1 -27162.912,E2 -27162.912} C_VEL
LIN {X 0,Y 107.427,Z 792.697,A -85,B 0,C 180,E1 -27166.958,E2 -27166.958} C_VEL
LIN {X 0,Y 104.458,Z 794.388,A -85,B 0,C 180,E1 -27177.635,E2 -27177.635} C_VEL
LIN {X 0,Y 104.358,Z 794.344,A -85,B 0,C 180,E1 -27179.83,E2 -27179.83} C_VEL
LIN {X 0,Y 105.082,Z 795.213,A -85,B 0,C 180,E1 -27187.446,E2 -27187.446} C_VEL
LIN {X 0,Y 106.466,Z 798.593,A -85,B 0,C 180,E1 -27192.995,E2 -27192.995} C_VEL
LIN {X 0,Y 108.343,Z 800.361,A -85,B 0,C 180,E1 -27197.216,E2 -27197.216} C_VEL
LIN {X 0,Y 110.409,Z 803.854,A -85,B 0,C 180,E1 -27201.066,E2 -27201.066} C_VEL
LIN {X 0,Y 111.607,Z 805.35,A -85,B 0,C 180,E1 -27202.872,E2 -27202.872} C_VEL
LIN {X 0,Y 114.623,Z 809.942,A -85,B 0,C 180,E1 -27206.885,E2 -27206.885} C_VEL
LIN {X 0,Y 117.773,Z 815.057,A -85,B 0,C 180,E1 -27210.406,E2 -27210.406} C_VEL
LIN {X 0,Y 121.434,Z 821.607,A -85,B 0,C 180,E1 -27213.946,E2 -27213.946} C_VEL
LIN {X 0,Y 125.395,Z 829.851,A -85,B 0,C 180,E1 -27217.343,E2 -27217.343} C_VEL
LIN {X 0,Y 123.868,Z 844.752,A -85,B 0,C 180,E1 -27218.194,E2 -27218.194} C_VEL
LIN {X 0,Y 121.678,Z 855.563,A -85,B 0,C 180,E1 -27219.267,E2 -27219.267} C_VEL
LIN {X 0,Y 119.007,Z 864.76,A -85,B 0,C 180,E1 -27220.513,E2 -27220.513} C_VEL
LIN {X 0,Y 116.231,Z 872.827,A -85,B 0,C 180,E1 -27222.075,E2 -27222.075} C_VEL
LIN {X 0,Y 113.257,Z 879.992,A -85,B 0,C 180,E1 -27223.832,E2 -27223.832} C_VEL
LIN {X 0,Y 109.271,Z 887.888,A -85,B 0,C 180,E1 -27226.258,E2 -27226.258} C_VEL
LIN {X 0,Y 105.06,Z 895.247,A -85,B 0,C 180,E1 -27229.29,E2 -27229.29} C_VEL
LIN {X 0,Y 100.13,Z 902.705,A -85,B 0,C 180,E1 -27233.373,E2 -27233.373} C_VEL
LIN {X 0,Y 94.987,Z 909.53,A -85,B 0,C 180,E1 -27238.807,E2 -27238.807} C_VEL
LIN {X 0,Y 90.746,Z 914.691,A -85,B 0,C 180,E1 -27244.789,E2 -27244.789} C_VEL
LIN {X 0,Y 88.461,Z 917.333,A -85,B 0,C 180,E1 -27249.053,E2 -27249.053} C_VEL
LIN {X 0,Y 85.913,Z 920.225,A -85,B 0,C 180,E1 -27255.794,E2 -27255.794} C_VEL
LIN {X 0,Y 84.803,Z 921.482,A -85,B 0,C 180,E1 -27260.459,E2 -27260.459} C_VEL
LIN {X 0,Y 84.201,Z 922.27,A -85,B 0,C 180,E1 -27265.212,E2 -27265.212} C_VEL
LIN {X 0,Y 84.024,Z 922.569,A -85,B 0,C 180,E1 -27270,E2 -27270} C_VEL
LIN {X 0,Y 84.163,Z 922.289,A -85,B 0,C 180,E1 -27274.79,E2 -27274.79} C_VEL
LIN {X 0,Y 84.802,Z 921.536,A -85,B 0,C 180,E1 -27279.541,E2 -27279.541} C_VEL
LIN {X 0,Y 85.901,Z 920.316,A -85,B 0,C 180,E1 -27284.208,E2 -27284.208} C_VEL
LIN {X 0,Y 88.42,Z 917.462,A -85,B 0,C 180,E1 -27290.958,E2 -27290.958} C_VEL
LIN {X 0,Y 90.657,Z 914.862,A -85,B 0,C 180,E1 -27295.238,E2 -27295.238} C_VEL
LIN {X 0,Y 94.96,Z 909.745,A -85,B 0,C 180,E1 -27301.203,E2 -27301.203} C_VEL
LIN {X 0,Y 99.19,Z 904.238,A -85,B 0,C 180,E1 -27305.771,E2 -27305.771} C_VEL
LIN {X 0,Y 103.942,Z 897.309,A -85,B 0,C 180,E1 -27309.966,E2 -27309.966} C_VEL
LIN {X 0,Y 108.669,Z 889.35,A -85,B 0,C 180,E1 -27313.405,E2 -27313.405} C_VEL
LIN {X 0,Y 112.605,Z 881.759,A -85,B 0,C 180,E1 -27315.869,E2 -27315.869} C_VEL
LIN {X 0,Y 116.101,Z 873.72,A -85,B 0,C 180,E1 -27317.895,E2 -27317.895} C_VEL
LIN {X 0,Y 119.235,Z 865.018,A -85,B 0,C 180,E1 -27319.553,E2 -27319.553} C_VEL
LIN {X 0,Y 121.82,Z 855.795,A -85,B 0,C 180,E1 -27320.875,E2 -27320.875} C_VEL
LIN {X 0,Y 124.005,Z 844.754,A -85,B 0,C 180,E1 -27322.014,E2 -27322.014} C_VEL
LIN {X 0,Y 125.595,Z 829.983,A -85,B 0,C 180,E1 -27322.816,E2 -27322.816} C_VEL
LIN {X 0,Y 121.269,Z 821.141,A -85,B 0,C 180,E1 -27326.544,E2 -27326.544} C_VEL
LIN {X 0,Y 117.463,Z 814.414,A -85,B 0,C 180,E1 -27330.298,E2 -27330.298} C_VEL
LIN {X 0,Y 113.755,Z 808.381,A -85,B 0,C 180,E1 -27334.65,E2 -27334.65} C_VEL
LIN {X 0,Y 111.205,Z 804.536,A -85,B 0,C 180,E1 -27338.262,E2 -27338.262} C_VEL
LIN {X 0,Y 108.831,Z 801.273,A -85,B 0,C 180,E1 -27342.379,E2 -27342.379} C_VEL
LIN {X 0,Y 108.329,Z 800.116,A -85,B 0,C 180,E1 -27343.51,E2 -27343.51} C_VEL
LIN {X 0,Y 106.124,Z 797.877,A -85,B 0,C 180,E1 -27349.024,E2 -27349.024} C_VEL
LIN {X 0,Y 105.161,Z 795.208,A -85,B 0,C 180,E1 -27353.765,E2 -27353.765} C_VEL
LIN {X 0,Y 104.665,Z 794.475,A -85,B 0,C 180,E1 -27360,E2 -27360} C_VEL
LIN {X 0,Y 105.226,Z 795.352,A -85,B 0,C 180,E1 -27366.279,E2 -27366.279} C_VEL
LIN {X 0,Y 107.224,Z 799.308,A -85,B 0,C 180,E1 -27373.744,E2 -27373.744} C_VEL
LIN {X 0,Y 108.533,Z 800.533,A -85,B 0,C 180,E1 -27376.578,E2 -27376.578} C_VEL
LIN {X 0,Y 110.831,Z 804.198,A -85,B 0,C 180,E1 -27380.813,E2 -27380.813} C_VEL
LIN {X 0,Y 111.811,Z 805.452,A -85,B 0,C 180,E1 -27382.293,E2 -27382.293} C_VEL
LIN {X 0,Y 114.731,Z 809.924,A -85,B 0,C 180,E1 -27386.213,E2 -27386.213} C_VEL
LIN {X 0,Y 117.641,Z 814.639,A -85,B 0,C 180,E1 -27389.513,E2 -27389.513} C_VEL
LIN {X 0,Y 121.073,Z 820.86,A -85,B 0,C 180,E1 -27392.916,E2 -27392.916} C_VEL
LIN {X 0,Y 124.131,Z 829.352,A -85,B 0,C 180,E1 -27395.848,E2 -27395.848} C_VEL
LIN {X 0,Y 125.28,Z 833.009,A -85,B 0,C 180,E1 -27396.906,E2 -27396.906} C_VEL
LIN {X 0,Y 123.751,Z 848.569,A -85,B 0,C 180,E1 -27397.761,E2 -27397.761} C_VEL
LIN {X 0,Y 121.662,Z 858.905,A -85,B 0,C 180,E1 -27398.7,E2 -27398.7} C_VEL
LIN {X 0,Y 119.012,Z 868.076,A -85,B 0,C 180,E1 -27399.853,E2 -27399.853} C_VEL
LIN {X 0,Y 115.932,Z 876.738,A -85,B 0,C 180,E1 -27401.393,E2 -27401.393} C_VEL
LIN {X 0,Y 112.366,Z 885.025,A -85,B 0,C 180,E1 -27403.359,E2 -27403.359} C_VEL
LIN {X 0,Y 108.367,Z 892.867,A -85,B 0,C 180,E1 -27405.799,E2 -27405.799} C_VEL
LIN {X 0,Y 104.041,Z 900.207,A -85,B 0,C 180,E1 -27408.805,E2 -27408.805} C_VEL
LIN {X 0,Y 99.108,Z 907.656,A -85,B 0,C 180,E1 -27412.932,E2 -27412.932} C_VEL
LIN {X 0,Y 94.67,Z 913.492,A -85,B 0,C 180,E1 -27417.438,E2 -27417.438} C_VEL
LIN {X 0,Y 90.899,Z 918.099,A -85,B 0,C 180,E1 -27422.361,E2 -27422.361} C_VEL
LIN {X 0,Y 88.548,Z 921.101,A -85,B 0,C 180,E1 -27426.619,E2 -27426.619} C_VEL
LIN {X 0,Y 86.637,Z 923.433,A -85,B 0,C 180,E1 -27431.066,E2 -27431.066} C_VEL
LIN {X 0,Y 85.203,Z 925.181,A -85,B 0,C 180,E1 -27435.673,E2 -27435.673} C_VEL
LIN {X 0,Y 84.301,Z 926.434,A -85,B 0,C 180,E1 -27440.402,E2 -27440.402} C_VEL
LIN {X 0,Y 83.877,Z 927.213,A -85,B 0,C 180,E1 -27445.194,E2 -27445.194} C_VEL
LIN {X 0,Y 83.885,Z 927.51,A -85,B 0,C 180,E1 -27450,E2 -27450} C_VEL
LIN {X 0,Y 83.873,Z 927.201,A -85,B 0,C 180,E1 -27454.807,E2 -27454.807} C_VEL
LIN {X 0,Y 84.286,Z 926.397,A -85,B 0,C 180,E1 -27459.6,E2 -27459.6} C_VEL
LIN {X 0,Y 85.203,Z 925.12,A -85,B 0,C 180,E1 -27464.327,E2 -27464.327} C_VEL
LIN {X 0,Y 87.51,Z 922.186,A -85,B 0,C 180,E1 -27471.186,E2 -27471.186} C_VEL
LIN {X 0,Y 89.651,Z 919.514,A -85,B 0,C 180,E1 -27475.541,E2 -27475.541} C_VEL
LIN {X 0,Y 93.873,Z 914.308,A -85,B 0,C 180,E1 -27481.606,E2 -27481.606} C_VEL
LIN {X 0,Y 99.075,Z 907.445,A -85,B 0,C 180,E1 -27487.082,E2 -27487.082} C_VEL
LIN {X 0,Y 104.034,Z 899.954,A -85,B 0,C 180,E1 -27491.198,E2 -27491.198} C_VEL
LIN {X 0,Y 108.366,Z 892.568,A -85,B 0,C 180,E1 -27494.202,E2 -27494.202} C_VEL
LIN {X 0,Y 112.405,Z 884.606,A -85,B 0,C 180,E1 -27496.649,E2 -27496.649} C_VEL
LIN {X 0,Y 116.515,Z 874.783,A -85,B 0,C 180,E1 -27498.936,E2 -27498.936} C_VEL
LIN {X 0,Y 120.035,Z 864.232,A -85,B 0,C 180,E1 -27500.598,E2 -27500.598} C_VEL
LIN {X 0,Y 122.593,Z 853.686,A -85,B 0,C 180,E1 -27501.722,E2 -27501.722} C_VEL
LIN {X 0,Y 124.131,Z 843.912,A -85,B 0,C 180,E1 -27502.434,E2 -27502.434} C_VEL
LIN {X 0,Y 125.084,Z 832.837,A -85,B 0,C 180,E1 -27503.026,E2 -27503.026} C_VEL
LIN {X 0,Y 121.972,Z 823.473,A -85,B 0,C 180,E1 -27505.945,E2 -27505.945} C_VEL
LIN {X 0,Y 119.835,Z 818.603,A -85,B 0,C 180,E1 -27508.006,E2 -27508.006} C_VEL
LIN {X 0,Y 115.945,Z 811.935,A -85,B 0,C 180,E1 -27512.043,E2 -27512.043} C_VEL
LIN {X 0,Y 113.446,Z 808.088,A -85,B 0,C 180,E1 -27515.052,E2 -27515.052} C_VEL
LIN {X 0,Y 111.062,Z 804.473,A -85,B 0,C 180,E1 -27518.419,E2 -27518.419} C_VEL
LIN {X 0,Y 108.643,Z 801.025,A -85,B 0,C 180,E1 -27522.592,E2 -27522.592} C_VEL
LIN {X 0,Y 108.002,Z 799.936,A -85,B 0,C 180,E1 -27523.945,E2 -27523.945} C_VEL
LIN {X 0,Y 105.966,Z 797.729,A -85,B 0,C 180,E1 -27529.008,E2 -27529.008} C_VEL
LIN {X 0,Y 105.036,Z 795.1,A -85,B 0,C 180,E1 -27533.276,E2 -27533.276} C_VEL
LIN {X 0,Y 104.358,Z 794.344,A -85,B 0,C 180,E1 -27539.83,E2 -27539.83} C_VEL
LIN {X 0,Y 104.321,Z 795,A -85,B 0,C 180,E1 -27541.929,E2 -27541.929} C_VEL
LIN {X 0,Y 104.259,Z 796.837,A -85,B 0,C 180,E1 -27543.863,E2 -27543.863} C_VEL
LIN {X 0,Y 104.417,Z 803.276,A -85,B 0,C 180,E1 -27548.769,E2 -27548.769} C_VEL
LIN {X 0,Y 104.687,Z 804.376,A -85,B 0,C 180,E1 -27550.143,E2 -27550.143} C_VEL
LIN {X 0,Y 106.916,Z 807.198,A -85,B 0,C 180,E1 -27556.223,E2 -27556.223} C_VEL
LIN {X 0,Y 109.241,Z 810.979,A -85,B 0,C 180,E1 -27560.744,E2 -27560.744} C_VEL
LIN {X 0,Y 112.457,Z 816.192,A -85,B 0,C 180,E1 -27565.526,E2 -27565.526} C_VEL
LIN {X 0,Y 115.713,Z 821.748,A -85,B 0,C 180,E1 -27569.447,E2 -27569.447} C_VEL
LIN {X 0,Y 119.873,Z 830.082,A -85,B 0,C 180,E1 -27573.723,E2 -27573.723} C_VEL
LIN {X 0,Y 120.987,Z 832.587,A -85,B 0,C 180,E1 -27574.77,E2 -27574.77} C_VEL
LIN {X 0,Y 119.383,Z 846.198,A -85,B 0,C 180,E1 -27575.636,E2 -27575.636} C_VEL
LIN {X 0,Y 117.356,Z 855.684,A -85,B 0,C 180,E1 -27576.582,E2 -27576.582} C_VEL
LIN {X 0,Y 114.48,Z 865.144,A -85,B 0,C 180,E1 -27577.85,E2 -27577.85} C_VEL
LIN {X 0,Y 111.466,Z 873.382,A -85,B 0,C 180,E1 -27579.448,E2 -27579.448} C_VEL
LIN {X 0,Y 108.477,Z 880.204,A -85,B 0,C 180,E1 -27581.135,E2 -27581.135} C_VEL
LIN {X 0,Y 104.274,Z 888.099,A -85,B 0,C 180,E1 -27583.569,E2 -27583.569} C_VEL
LIN {X 0,Y 99.799,Z 895.459,A -85,B 0,C 180,E1 -27586.638,E2 -27586.638} C_VEL
LIN {X 0,Y 94.538,Z 902.916,A -85,B 0,C 180,E1 -27590.81,E2 -27590.81} C_VEL
LIN {X 0,Y 89,Z 909.74,A -85,B 0,C 180,E1 -27596.443,E2 -27596.443} C_VEL
LIN {X 0,Y 84.369,Z 914.901,A -85,B 0,C 180,E1 -27602.732,E2 -27602.732} C_VEL
LIN {X 0,Y 81.879,Z 917.543,A -85,B 0,C 180,E1 -27607.278,E2 -27607.278} C_VEL
LIN {X 0,Y 79.058,Z 920.435,A -85,B 0,C 180,E1 -27614.533,E2 -27614.533} C_VEL
LIN {X 0,Y 77.829,Z 921.691,A -85,B 0,C 180,E1 -27619.595,E2 -27619.595} C_VEL
LIN {X 0,Y 77.127,Z 922.479,A -85,B 0,C 180,E1 -27624.772,E2 -27624.772} C_VEL
LIN {X 0,Y 76.927,Z 922.778,A -85,B 0,C 180,E1 -27630,E2 -27630} C_VEL
LIN {X 0,Y 77.096,Z 922.498,A -85,B 0,C 180,E1 -27635.23,E2 -27635.23} C_VEL
LIN {X 0,Y 77.828,Z 921.744,A -85,B 0,C 180,E1 -27640.405,E2 -27640.405} C_VEL
LIN {X 0,Y 79.046,Z 920.524,A -85,B 0,C 180,E1 -27645.47,E2 -27645.47} C_VEL
LIN {X 0,Y 81.839,Z 917.67,A -85,B 0,C 180,E1 -27652.733,E2 -27652.733} C_VEL
LIN {X 0,Y 84.287,Z 915.069,A -85,B 0,C 180,E1 -27657.297,E2 -27657.297} C_VEL
LIN {X 0,Y 88.974,Z 909.952,A -85,B 0,C 180,E1 -27663.568,E2 -27663.568} C_VEL
LIN {X 0,Y 93.523,Z 904.445,A -85,B 0,C 180,E1 -27668.314,E2 -27668.314} C_VEL
LIN {X 0,Y 98.621,Z 897.514,A -85,B 0,C 180,E1 -27672.61,E2 -27672.61} C_VEL
LIN {X 0,Y 103.633,Z 889.555,A -85,B 0,C 180,E1 -27676.1,E2 -27676.1} C_VEL
LIN {X 0,Y 107.792,Z 881.963,A -85,B 0,C 180,E1 -27678.573,E2 -27678.573} C_VEL
LIN {X 0,Y 110.949,Z 875.186,A -85,B 0,C 180,E1 -27680.327,E2 -27680.327} C_VEL
LIN {X 0,Y 114.127,Z 867.091,A -85,B 0,C 180,E1 -27681.94,E2 -27681.94} C_VEL
LIN {X 0,Y 116.966,Z 858.007,A -85,B 0,C 180,E1 -27683.294,E2 -27683.294} C_VEL
LIN {X 0,Y 118.947,Z 849.389,A -85,B 0,C 180,E1 -27684.274,E2 -27684.274} C_VEL
LIN {X 0,Y 120.426,Z 840.259,A -85,B 0,C 180,E1 -27684.97,E2 -27684.97} C_VEL
LIN {X 0,Y 121.199,Z 832.822,A -85,B 0,C 180,E1 -27685.377,E2 -27685.377} C_VEL
LIN {X 0,Y 117.402,Z 824.86,A -85,B 0,C 180,E1 -27689.102,E2 -27689.102} C_VEL
LIN {X 0,Y 113.959,Z 818.44,A -85,B 0,C 180,E1 -27693.02,E2 -27693.02} C_VEL
LIN {X 0,Y 111.368,Z 814.226,A -85,B 0,C 180,E1 -27696.456,E2 -27696.456} C_VEL
LIN {X 0,Y 109.411,Z 811.009,A -85,B 0,C 180,E1 -27699.544,E2 -27699.544} C_VEL
LIN {X 0,Y 107.107,Z 807.398,A -85,B 0,C 180,E1 -27704.051,E2 -27704.051} C_VEL
LIN {X 0,Y 106.594,Z 806.682,A -85,B 0,C 180,E1 -27705.246,E2 -27705.246} C_VEL
LIN {X 0,Y 104.706,Z 804.056,A -85,B 0,C 180,E1 -27711.07,E2 -27711.07} C_VEL
LIN {X 0,Y 104.218,Z 802.199,A -85,B 0,C 180,E1 -27714.194,E2 -27714.194} C_VEL
LIN {X 0,Y 103.799,Z 801.53,A -85,B 0,C 180,E1 -27720,E2 -27720} C_VEL
LIN {X 0,Y 104.258,Z 802.423,A -85,B 0,C 180,E1 -27725.803,E2 -27725.803} C_VEL
LIN {X 0,Y 105.827,Z 805.924,A -85,B 0,C 180,E1 -27732.464,E2 -27732.464} C_VEL
LIN {X 0,Y 107.08,Z 807.253,A -85,B 0,C 180,E1 -27735.494,E2 -27735.494} C_VEL
LIN {X 0,Y 109.312,Z 810.921,A -85,B 0,C 180,E1 -27739.929,E2 -27739.929} C_VEL
LIN {X 0,Y 112.549,Z 816.074,A -85,B 0,C 180,E1 -27744.805,E2 -27744.805} C_VEL
LIN {X 0,Y 115.903,Z 821.928,A -85,B 0,C 180,E1 -27748.894,E2 -27748.894} C_VEL
LIN {X 0,Y 118.081,Z 826.441,A -85,B 0,C 180,E1 -27751.26,E2 -27751.26} C_VEL
LIN {X 0,Y 120.566,Z 834.04,A -85,B 0,C 180,E1 -27753.94,E2 -27753.94} C_VEL
LIN {X 0,Y 120.938,Z 835.306,A -85,B 0,C 180,E1 -27754.33,E2 -27754.33} C_VEL
LIN {X 0,Y 119.406,Z 849.144,A -85,B 0,C 180,E1 -27755.137,E2 -27755.137} C_VEL
LIN {X 0,Y 117.048,Z 859.828,A -85,B 0,C 180,E1 -27756.127,E2 -27756.127} C_VEL
LIN {X 0,Y 114.602,Z 867.873,A -85,B 0,C 180,E1 -27757.133,E2 -27757.133} C_VEL
LIN {X 0,Y 111.355,Z 876.533,A -85,B 0,C 180,E1 -27758.645,E2 -27758.645} C_VEL
LIN {X 0,Y 108.099,Z 883.83,A -85,B 0,C 180,E1 -27760.333,E2 -27760.333} C_VEL
LIN {X 0,Y 104.565,Z 890.615,A -85,B 0,C 180,E1 -27762.325,E2 -27762.325} C_VEL
LIN {X 0,Y 99.924,Z 898.292,A -85,B 0,C 180,E1 -27765.305,E2 -27765.305} C_VEL
LIN {X 0,Y 95.525,Z 904.61,A -85,B 0,C 180,E1 -27768.536,E2 -27768.536} C_VEL
LIN {X 0,Y 91.549,Z 909.864,A -85,B 0,C 180,E1 -27772.11,E2 -27772.11} C_VEL
LIN {X 0,Y 87.888,Z 914.245,A -85,B 0,C 180,E1 -27775.961,E2 -27775.961} C_VEL
LIN {X 0,Y 83.276,Z 919.418,A -85,B 0,C 180,E1 -27782.344,E2 -27782.344} C_VEL
LIN {X 0,Y 79.921,Z 923.224,A -85,B 0,C 180,E1 -27789.406,E2 -27789.406} C_VEL
LIN {X 0,Y 78.323,Z 924.972,A -85,B 0,C 180,E1 -27794.384,E2 -27794.384} C_VEL
LIN {X 0,Y 77.296,Z 926.225,A -85,B 0,C 180,E1 -27799.523,E2 -27799.523} C_VEL
LIN {X 0,Y 76.799,Z 927.004,A -85,B 0,C 180,E1 -27804.749,E2 -27804.749} C_VEL
LIN {X 0,Y 76.784,Z 927.301,A -85,B 0,C 180,E1 -27810,E2 -27810} C_VEL
LIN {X 0,Y 76.796,Z 926.992,A -85,B 0,C 180,E1 -27815.251,E2 -27815.251} C_VEL
LIN {X 0,Y 77.284,Z 926.187,A -85,B 0,C 180,E1 -27820.479,E2 -27820.479} C_VEL
LIN {X 0,Y 78.322,Z 924.91,A -85,B 0,C 180,E1 -27825.616,E2 -27825.616} C_VEL
LIN {X 0,Y 80.911,Z 921.975,A -85,B 0,C 180,E1 -27833.009,E2 -27833.009} C_VEL
LIN {X 0,Y 83.275,Z 919.303,A -85,B 0,C 180,E1 -27837.657,E2 -27837.657} C_VEL
LIN {X 0,Y 87.887,Z 914.097,A -85,B 0,C 180,E1 -27844.04,E2 -27844.04} C_VEL
LIN {X 0,Y 93.479,Z 907.233,A -85,B 0,C 180,E1 -27849.721,E2 -27849.721} C_VEL
LIN {X 0,Y 98.808,Z 899.743,A -85,B 0,C 180,E1 -27853.907,E2 -27853.907} C_VEL
LIN {X 0,Y 102.986,Z 893.073,A -85,B 0,C 180,E1 -27856.688,E2 -27856.688} C_VEL
LIN {X 0,Y 106.782,Z 886.169,A -85,B 0,C 180,E1 -27858.903,E2 -27858.903} C_VEL
LIN {X 0,Y 110.716,Z 877.576,A -85,B 0,C 180,E1 -27861.042,E2 -27861.042} C_VEL
LIN {X 0,Y 113.925,Z 869.173,A -85,B 0,C 180,E1 -27862.585,E2 -27862.585} C_VEL
LIN {X 0,Y 116.847,Z 859.77,A -85,B 0,C 180,E1 -27863.801,E2 -27863.801} C_VEL
LIN {X 0,Y 119.269,Z 848.735,A -85,B 0,C 180,E1 -27864.816,E2 -27864.816} C_VEL
LIN {X 0,Y 120.762,Z 835.214,A -85,B 0,C 180,E1 -27865.574,E2 -27865.574} C_VEL
LIN {X 0,Y 118.224,Z 827.224,A -85,B 0,C 180,E1 -27868.283,E2 -27868.283} C_VEL
LIN {X 0,Y 116.582,Z 823.45,A -85,B 0,C 180,E1 -27870.052,E2 -27870.052} C_VEL
LIN {X 0,Y 113.123,Z 817.262,A -85,B 0,C 180,E1 -27874.077,E2 -27874.077} C_VEL
LIN {X 0,Y 111.227,Z 814.119,A -85,B 0,C 180,E1 -27876.634,E2 -27876.634} C_VEL
LIN {X 0,Y 109.166,Z 810.832,A -85,B 0,C 180,E1 -27879.847,E2 -27879.847} C_VEL
LIN {X 0,Y 106.878,Z 807.072,A -85,B 0,C 180,E1 -27884.338,E2 -27884.338} C_VEL
LIN {X 0,Y 104.557,Z 803.952,A -85,B 0,C 180,E1 -27890.906,E2 -27890.906} C_VEL
LIN {X 0,Y 103.994,Z 802.004,A -85,B 0,C 180,E1 -27894.182,E2 -27894.182} C_VEL
LIN {X 0,Y 103.495,Z 801.359,A -85,B 0,C 180,E1 -27900,E2 -27900} C_VEL
LIN {X 0,Y 104.066,Z 802.248,A -85,B 0,C 180,E1 -27906.788,E2 -27906.788} C_VEL
LIN {X 0,Y 104.687,Z 804.376,A -85,B 0,C 180,E1 -27910.143,E2 -27910.143} C_VEL
LIN {X 0,Y 105.464,Z 806.781,A -85,B 0,C 180,E1 -27913.064,E2 -27913.064} C_VEL
LIN {X 0,Y 106.889,Z 812.463,A -85,B 0,C 180,E1 -27917.39,E2 -27917.39} C_VEL
LIN {X 0,Y 108.302,Z 817.549,A -85,B 0,C 180,E1 -27920.634,E2 -27920.634} C_VEL
LIN {X 0,Y 110.234,Z 822.174,A -85,B 0,C 180,E1 -27923.928,E2 -27923.928} C_VEL
LIN {X 0,Y 113.13,Z 827.528,A -85,B 0,C 180,E1 -27927.802,E2 -27927.802} C_VEL
LIN {X 0,Y 116.714,Z 835.23,A -85,B 0,C 180,E1 -27931.898,E2 -27931.898} C_VEL
LIN {X 0,Y 116.73,Z 836.937,A -85,B 0,C 180,E1 -27932.148,E2 -27932.148} C_VEL
LIN {X 0,Y 115.155,Z 847.643,A -85,B 0,C 180,E1 -27932.885,E2 -27932.885} C_VEL
LIN {X 0,Y 112.972,Z 856.916,A -85,B 0,C 180,E1 -27933.808,E2 -27933.808} C_VEL
LIN {X 0,Y 110.205,Z 865.547,A -85,B 0,C 180,E1 -27934.971,E2 -27934.971} C_VEL
LIN {X 0,Y 107.365,Z 872.973,A -85,B 0,C 180,E1 -27936.38,E2 -27936.38} C_VEL
LIN {X 0,Y 103.958,Z 880.416,A -85,B 0,C 180,E1 -27938.196,E2 -27938.196} C_VEL
LIN {X 0,Y 99.526,Z 888.311,A -85,B 0,C 180,E1 -27940.614,E2 -27940.614} C_VEL
LIN {X 0,Y 94.776,Z 895.67,A -85,B 0,C 180,E1 -27943.697,E2 -27943.697} C_VEL
LIN {X 0,Y 89.164,Z 903.127,A -85,B 0,C 180,E1 -27947.934,E2 -27947.934} C_VEL
LIN {X 0,Y 83.174,Z 909.951,A -85,B 0,C 180,E1 -27953.738,E2 -27953.738} C_VEL
LIN {X 0,Y 78.12,Z 915.111,A -85,B 0,C 180,E1 -27960.343,E2 -27960.343} C_VEL
LIN {X 0,Y 75.395,Z 917.752,A -85,B 0,C 180,E1 -27965.199,E2 -27965.199} C_VEL
LIN {X 0,Y 72.259,Z 920.644,A -85,B 0,C 180,E1 -27973.035,E2 -27973.035} C_VEL
LIN {X 0,Y 70.859,Z 921.9,A -85,B 0,C 180,E1 -27978.559,E2 -27978.559} C_VEL
LIN {X 0,Y 70.076,Z 922.687,A -85,B 0,C 180,E1 -27984.244,E2 -27984.244} C_VEL
LIN {X 0,Y 69.855,Z 922.986,A -85,B 0,C 180,E1 -27990,E2 -27990} C_VEL
LIN {X 0,Y 70.055,Z 922.706,A -85,B 0,C 180,E1 -27995.758,E2 -27995.758} C_VEL
LIN {X 0,Y 70.857,Z 921.953,A -85,B 0,C 180,E1 -28001.442,E2 -28001.442} C_VEL
LIN {X 0,Y 72.247,Z 920.732,A -85,B 0,C 180,E1 -28006.968,E2 -28006.968} C_VEL
LIN {X 0,Y 75.331,Z 917.878,A -85,B 0,C 180,E1 -28014.824,E2 -28014.824} C_VEL
LIN {X 0,Y 78.048,Z 915.277,A -85,B 0,C 180,E1 -28019.687,E2 -28019.687} C_VEL
LIN {X 0,Y 83.147,Z 910.159,A -85,B 0,C 180,E1 -28026.276,E2 -28026.276} C_VEL
LIN {X 0,Y 88.071,Z 904.652,A -85,B 0,C 180,E1 -28031.174,E2 -28031.174} C_VEL
LIN {X 0,Y 93.535,Z 897.72,A -85,B 0,C 180,E1 -28035.546,E2 -28035.546} C_VEL
LIN {X 0,Y 98.85,Z 889.761,A -85,B 0,C 180,E1 -28039.061,E2 -28039.061} C_VEL
LIN {X 0,Y 103.245,Z 882.167,A -85,B 0,C 180,E1 -28041.519,E2 -28041.519} C_VEL
LIN {X 0,Y 107.152,Z 874.057,A -85,B 0,C 180,E1 -28043.539,E2 -28043.539} C_VEL
LIN {X 0,Y 110.547,Z 865.49,A -85,B 0,C 180,E1 -28045.137,E2 -28045.137} C_VEL
LIN {X 0,Y 113.189,Z 857.045,A -85,B 0,C 180,E1 -28046.325,E2 -28046.325} C_VEL
LIN {X 0,Y 115.422,Z 847.233,A -85,B 0,C 180,E1 -28047.353,E2 -28047.353} C_VEL
LIN {X 0,Y 117.046,Z 835.776,A -85,B 0,C 180,E1 -28048.122,E2 -28048.122} C_VEL
LIN {X 0,Y 113.817,Z 828.722,A -85,B 0,C 180,E1 -28051.778,E2 -28051.778} C_VEL
LIN {X 0,Y 110.71,Z 822.841,A -85,B 0,C 180,E1 -28055.87,E2 -28055.87} C_VEL
LIN {X 0,Y 108.934,Z 819.721,A -85,B 0,C 180,E1 -28058.62,E2 -28058.62} C_VEL
LIN {X 0,Y 107.494,Z 817.25,A -85,B 0,C 180,E1 -28061.197,E2 -28061.197} C_VEL
LIN {X 0,Y 105.312,Z 813.493,A -85,B 0,C 180,E1 -28066.148,E2 -28066.148} C_VEL
LIN {X 0,Y 103.579,Z 810.757,A -85,B 0,C 180,E1 -28072.2,E2 -28072.2} C_VEL
LIN {X 0,Y 103.225,Z 809.107,A -85,B 0,C 180,E1 -28075.049,E2 -28075.049} C_VEL
LIN {X 0,Y 102.943,Z 808.674,A -85,B 0,C 180,E1 -28080.978,E2 -28080.978} C_VEL
LIN {X 0,Y 103.268,Z 809.308,A -85,B 0,C 180,E1 -28085.014,E2 -28085.014} C_VEL
LIN {X 0,Y 104.636,Z 812.748,A -85,B 0,C 180,E1 -28091.624,E2 -28091.624} C_VEL
LIN {X 0,Y 105.687,Z 814.04,A -85,B 0,C 180,E1 -28094.44,E2 -28094.44} C_VEL
LIN {X 0,Y 108.257,Z 818.486,A -85,B 0,C 180,E1 -28099.833,E2 -28099.833} C_VEL
LIN {X 0,Y 110.479,Z 822.352,A -85,B 0,C 180,E1 -28103.411,E2 -28103.411} C_VEL
LIN {X 0,Y 113.339,Z 827.713,A -85,B 0,C 180,E1 -28107.26,E2 -28107.26} C_VEL
LIN {X 0,Y 115.157,Z 831.903,A -85,B 0,C 180,E1 -28109.475,E2 -28109.475} C_VEL
LIN {X 0,Y 116.897,Z 837.698,A -85,B 0,C 180,E1 -28111.608,E2 -28111.608} C_VEL
LIN {X 0,Y 115.131,Z 850.492,A -85,B 0,C 180,E1 -28112.371,E2 -28112.371} C_VEL
LIN {X 0,Y 113.01,Z 859.627,A -85,B 0,C 180,E1 -28113.22,E2 -28113.22} C_VEL
LIN {X 0,Y 109.777,Z 869.545,A -85,B 0,C 180,E1 -28114.486,E2 -28114.486} C_VEL
LIN {X 0,Y 106.411,Z 877.832,A -85,B 0,C 180,E1 -28115.996,E2 -28115.996} C_VEL
LIN {X 0,Y 102.231,Z 886.334,A -85,B 0,C 180,E1 -28118.08,E2 -28118.08} C_VEL
LIN {X 0,Y 96.97,Z 895.273,A -85,B 0,C 180,E1 -28121.063,E2 -28121.063} C_VEL
LIN {X 0,Y 91.475,Z 902.981,A -85,B 0,C 180,E1 -28124.71,E2 -28124.71} C_VEL
LIN {X 0,Y 87.096,Z 908.48,A -85,B 0,C 180,E1 -28128.263,E2 -28128.263} C_VEL
LIN {X 0,Y 82.087,Z 914.037,A -85,B 0,C 180,E1 -28133.179,E2 -28133.179} C_VEL
LIN {X 0,Y 77.04,Z 919.21,A -85,B 0,C 180,E1 -28139.885,E2 -28139.885} C_VEL
LIN {X 0,Y 73.29,Z 923.015,A -85,B 0,C 180,E1 -28147.445,E2 -28147.445} C_VEL
LIN {X 0,Y 71.498,Z 924.763,A -85,B 0,C 180,E1 -28152.849,E2 -28152.849} C_VEL
LIN {X 0,Y 70.324,Z 926.016,A -85,B 0,C 180,E1 -28158.47,E2 -28158.47} C_VEL
LIN {X 0,Y 69.744,Z 926.796,A -85,B 0,C 180,E1 -28164.217,E2 -28164.217} C_VEL
LIN {X 0,Y 69.705,Z 927.093,A -85,B 0,C 180,E1 -28170,E2 -28170} C_VEL
LIN {X 0,Y 69.74,Z 926.783,A -85,B 0,C 180,E1 -28175.784,E2 -28175.784} C_VEL
LIN {X 0,Y 70.315,Z 925.978,A -85,B 0,C 180,E1 -28181.531,E2 -28181.531} C_VEL
LIN {X 0,Y 71.498,Z 924.7,A -85,B 0,C 180,E1 -28187.151,E2 -28187.151} C_VEL
LIN {X 0,Y 74.412,Z 921.765,A -85,B 0,C 180,E1 -28195.152,E2 -28195.152} C_VEL
LIN {X 0,Y 77.039,Z 919.093,A -85,B 0,C 180,E1 -28200.115,E2 -28200.115} C_VEL
LIN {X 0,Y 82.086,Z 913.886,A -85,B 0,C 180,E1 -28206.821,E2 -28206.821} C_VEL
LIN {X 0,Y 88.111,Z 907.021,A -85,B 0,C 180,E1 -28212.686,E2 -28212.686} C_VEL
LIN {X 0,Y 93.813,Z 899.531,A -85,B 0,C 180,E1 -28216.922,E2 -28216.922} C_VEL
LIN {X 0,Y 98.335,Z 892.702,A -85,B 0,C 180,E1 -28219.767,E2 -28219.767} C_VEL
LIN {X 0,Y 102.255,Z 885.956,A -85,B 0,C 180,E1 -28221.903,E2 -28221.903} C_VEL
LIN {X 0,Y 106.385,Z 877.362,A -85,B 0,C 180,E1 -28224.023,E2 -28224.023} C_VEL
LIN {X 0,Y 109.766,Z 868.959,A -85,B 0,C 180,E1 -28225.523,E2 -28225.523} C_VEL
LIN {X 0,Y 112.803,Z 859.554,A -85,B 0,C 180,E1 -28226.711,E2 -28226.711} C_VEL
LIN {X 0,Y 115.326,Z 848.553,A -85,B 0,C 180,E1 -28227.691,E2 -28227.691} C_VEL
LIN {X 0,Y 116.673,Z 837.472,A -85,B 0,C 180,E1 -28228.337,E2 -28228.337} C_VEL
LIN {X 0,Y 114.422,Z 830.188,A -85,B 0,C 180,E1 -28231.105,E2 -28231.105} C_VEL
LIN {X 0,Y 111.215,Z 823.852,A -85,B 0,C 180,E1 -28235.154,E2 -28235.154} C_VEL
LIN {X 0,Y 108.971,Z 819.925,A -85,B 0,C 180,E1 -28238.481,E2 -28238.481} C_VEL
LIN {X 0,Y 107.312,Z 817.133,A -85,B 0,C 180,E1 -28241.382,E2 -28241.382} C_VEL
LIN {X 0,Y 105.166,Z 813.424,A -85,B 0,C 180,E1 -28246.164,E2 -28246.164} C_VEL
LIN {X 0,Y 103.433,Z 810.719,A -85,B 0,C 180,E1 -28251.914,E2 -28251.914} C_VEL
LIN {X 0,Y 102.977,Z 808.928,A -85,B 0,C 180,E1 -28255.107,E2 -28255.107} C_VEL
LIN {X 0,Y 102.626,Z 808.508,A -85,B 0,C 180,E1 -28260.981,E2 -28260.981} C_VEL
LIN {X 0,Y 103.043,Z 809.105,A -85,B 0,C 180,E1 -28265.872,E2 -28265.872} C_VEL
LIN {X 0,Y 104.21,Z 812.401,A -85,B 0,C 180,E1 -28271.673,E2 -28271.673} C_VEL
LIN {X 0,Y 105.508,Z 813.97,A -85,B 0,C 180,E1 -28275.16,E2 -28275.16} C_VEL
LIN {X 0,Y 108.122,Z 818.551,A -85,B 0,C 180,E1 -28280.564,E2 -28280.564} C_VEL
LIN {X 0,Y 110.234,Z 822.174,A -85,B 0,C 180,E1 -28283.928,E2 -28283.928} C_VEL
LIN {X 0,Y 111.305,Z 824.677,A -85,B 0,C 180,E1 -28285.515,E2 -28285.515} C_VEL
LIN {X 0,Y 112.132,Z 827.802,A -85,B 0,C 180,E1 -28286.824,E2 -28286.824} C_VEL
LIN {X 0,Y 112.817,Z 832.613,A -85,B 0,C 180,E1 -28288.159,E2 -28288.159} C_VEL
LIN {X 0,Y 112.9,Z 837.879,A -85,B 0,C 180,E1 -28289.034,E2 -28289.034} C_VEL
LIN {X 0,Y 112.645,Z 840.598,A -85,B 0,C 180,E1 -28289.283,E2 -28289.283} C_VEL
LIN {X 0,Y 111.026,Z 849.827,A -85,B 0,C 180,E1 -28289.967,E2 -28289.967} C_VEL
LIN {X 0,Y 108.505,Z 859.418,A -85,B 0,C 180,E1 -28290.968,E2 -28290.968} C_VEL
LIN {X 0,Y 104.335,Z 870.872,A -85,B 0,C 180,E1 -28292.701,E2 -28292.701} C_VEL
LIN {X 0,Y 99.736,Z 880.628,A -85,B 0,C 180,E1 -28294.998,E2 -28294.998} C_VEL
LIN {X 0,Y 95.063,Z 888.523,A -85,B 0,C 180,E1 -28297.369,E2 -28297.369} C_VEL
LIN {X 0,Y 90.031,Z 895.881,A -85,B 0,C 180,E1 -28300.438,E2 -28300.438} C_VEL
LIN {X 0,Y 84.038,Z 903.337,A -85,B 0,C 180,E1 -28304.696,E2 -28304.696} C_VEL
LIN {X 0,Y 77.562,Z 910.161,A -85,B 0,C 180,E1 -28310.633,E2 -28310.633} C_VEL
LIN {X 0,Y 72.036,Z 915.322,A -85,B 0,C 180,E1 -28317.548,E2 -28317.548} C_VEL
LIN {X 0,Y 69.008,Z 917.962,A -85,B 0,C 180,E1 -28322.723,E2 -28322.723} C_VEL
LIN {X 0,Y 65.507,Z 920.853,A -85,B 0,C 180,E1 -28331.225,E2 -28331.225} C_VEL
LIN {X 0,Y 63.933,Z 922.109,A -85,B 0,C 180,E1 -28337.299,E2 -28337.299} C_VEL
LIN {X 0,Y 63.024,Z 922.896,A -85,B 0,C 180,E1 -28343.597,E2 -28343.597} C_VEL
LIN {X 0,Y 62.757,Z 923.195,A -85,B 0,C 180,E1 -28350,E2 -28350} C_VEL
LIN {X 0,Y 63.01,Z 922.914,A -85,B 0,C 180,E1 -28356.404,E2 -28356.404} C_VEL
LIN {X 0,Y 63.931,Z 922.161,A -85,B 0,C 180,E1 -28362.701,E2 -28362.701} C_VEL
LIN {X 0,Y 65.494,Z 920.94,A -85,B 0,C 180,E1 -28368.779,E2 -28368.779} C_VEL
LIN {X 0,Y 68.953,Z 918.086,A -85,B 0,C 180,E1 -28377.301,E2 -28377.301} C_VEL
LIN {X 0,Y 71.972,Z 915.484,A -85,B 0,C 180,E1 -28382.484,E2 -28382.484} C_VEL
LIN {X 0,Y 77.532,Z 910.367,A -85,B 0,C 180,E1 -28389.385,E2 -28389.385} C_VEL
LIN {X 0,Y 82.871,Z 904.858,A -85,B 0,C 180,E1 -28394.399,E2 -28394.399} C_VEL
LIN {X 0,Y 88.721,Z 897.926,A -85,B 0,C 180,E1 -28398.811,E2 -28398.811} C_VEL
LIN {X 0,Y 94.358,Z 889.966,A -85,B 0,C 180,E1 -28402.314,E2 -28402.314} C_VEL
LIN {X 0,Y 98.996,Z 882.372,A -85,B 0,C 180,E1 -28404.728,E2 -28404.728} C_VEL
LIN {X 0,Y 103.162,Z 874.124,A -85,B 0,C 180,E1 -28406.736,E2 -28406.736} C_VEL
LIN {X 0,Y 106.69,Z 865.602,A -85,B 0,C 180,E1 -28408.276,E2 -28408.276} C_VEL
LIN {X 0,Y 109.571,Z 856.693,A -85,B 0,C 180,E1 -28409.487,E2 -28409.487} C_VEL
LIN {X 0,Y 112.101,Z 845.753,A -85,B 0,C 180,E1 -28410.564,E2 -28410.564} C_VEL
LIN {X 0,Y 113.103,Z 838.839,A -85,B 0,C 180,E1 -28410.995,E2 -28410.995} C_VEL
LIN {X 0,Y 110.357,Z 832.405,A -85,B 0,C 180,E1 -28414.804,E2 -28414.804} C_VEL
LIN {X 0,Y 107.528,Z 826.765,A -85,B 0,C 180,E1 -28419.288,E2 -28419.288} C_VEL
LIN {X 0,Y 105.833,Z 823.665,A -85,B 0,C 180,E1 -28422.581,E2 -28422.581} C_VEL
LIN {X 0,Y 104.092,Z 820.333,A -85,B 0,C 180,E1 -28426.977,E2 -28426.977} C_VEL
LIN {X 0,Y 102.512,Z 817.53,A -85,B 0,C 180,E1 -28433.224,E2 -28433.224} C_VEL
LIN {X 0,Y 102.239,Z 816.022,A -85,B 0,C 180,E1 -28436.058,E2 -28436.058} C_VEL
LIN {X 0,Y 102.076,Z 815.73,A -85,B 0,C 180,E1 -28440.986,E2 -28440.986} C_VEL
LIN {X 0,Y 102.295,Z 816.234,A -85,B 0,C 180,E1 -28444.22,E2 -28444.22} C_VEL
LIN {X 0,Y 103.465,Z 819.589,A -85,B 0,C 180,E1 -28450.766,E2 -28450.766} C_VEL
LIN {X 0,Y 104.385,Z 820.908,A -85,B 0,C 180,E1 -28453.505,E2 -28453.505} C_VEL
LIN {X 0,Y 106.545,Z 824.935,A -85,B 0,C 180,E1 -28458.508,E2 -28458.508} C_VEL
LIN {X 0,Y 108.59,Z 828.824,A -85,B 0,C 180,E1 -28462.145,E2 -28462.145} C_VEL
LIN {X 0,Y 111.127,Z 834.009,A -85,B 0,C 180,E1 -28465.898,E2 -28465.898} C_VEL
LIN {X 0,Y 112.275,Z 837.142,A -85,B 0,C 180,E1 -28467.495,E2 -28467.495} C_VEL
LIN {X 0,Y 113.063,Z 840.246,A -85,B 0,C 180,E1 -28468.692,E2 -28468.692} C_VEL
LIN {X 0,Y 111.433,Z 850.604,A -85,B 0,C 180,E1 -28469.321,E2 -28469.321} C_VEL
LIN {X 0,Y 109.396,Z 859.054,A -85,B 0,C 180,E1 -28470.067,E2 -28470.067} C_VEL
LIN {X 0,Y 106.649,Z 867.468,A -85,B 0,C 180,E1 -28471.054,E2 -28471.054} C_VEL
LIN {X 0,Y 103.083,Z 876.124,A -85,B 0,C 180,E1 -28472.467,E2 -28472.467} C_VEL
LIN {X 0,Y 98.952,Z 884.405,A -85,B 0,C 180,E1 -28474.344,E2 -28474.344} C_VEL
LIN {X 0,Y 94.468,Z 891.91,A -85,B 0,C 180,E1 -28476.598,E2 -28476.598} C_VEL
LIN {X 0,Y 90.384,Z 897.88,A -85,B 0,C 180,E1 -28478.961,E2 -28478.961} C_VEL
LIN {X 0,Y 85.405,Z 904.197,A -85,B 0,C 180,E1 -28482.216,E2 -28482.216} C_VEL
LIN {X 0,Y 80.787,Z 909.449,A -85,B 0,C 180,E1 -28485.897,E2 -28485.897} C_VEL
LIN {X 0,Y 76.514,Z 913.829,A -85,B 0,C 180,E1 -28489.987,E2 -28489.987} C_VEL
LIN {X 0,Y 70.977,Z 919.002,A -85,B 0,C 180,E1 -28497.003,E2 -28497.003} C_VEL
LIN {X 0,Y 66.771,Z 922.807,A -85,B 0,C 180,E1 -28505.101,E2 -28505.101} C_VEL
LIN {X 0,Y 64.743,Z 924.555,A -85,B 0,C 180,E1 -28510.995,E2 -28510.995} C_VEL
LIN {X 0,Y 63.367,Z 925.807,A -85,B 0,C 180,E1 -28517.184,E2 -28517.184} C_VEL
LIN {X 0,Y 62.67,Z 926.586,A -85,B 0,C 180,E1 -28523.561,E2 -28523.561} C_VEL
LIN {X 0,Y 62.617,Z 926.884,A -85,B 0,C 180,E1 -28530,E2 -28530} C_VEL
LIN {X 0,Y 62.666,Z 926.573,A -85,B 0,C 180,E1 -28536.439,E2 -28536.439} C_VEL
LIN {X 0,Y 63.359,Z 925.768,A -85,B 0,C 180,E1 -28542.817,E2 -28542.817} C_VEL
LIN {X 0,Y 64.743,Z 924.49,A -85,B 0,C 180,E1 -28549.006,E2 -28549.006} C_VEL
LIN {X 0,Y 68.039,Z 921.555,A -85,B 0,C 180,E1 -28557.699,E2 -28557.699} C_VEL
LIN {X 0,Y 70.976,Z 918.882,A -85,B 0,C 180,E1 -28562.998,E2 -28562.998} C_VEL
LIN {X 0,Y 76.513,Z 913.675,A -85,B 0,C 180,E1 -28570.014,E2 -28570.014} C_VEL
LIN {X 0,Y 83.018,Z 906.809,A -85,B 0,C 180,E1 -28576.02,E2 -28576.02} C_VEL
LIN {X 0,Y 89.111,Z 899.319,A -85,B 0,C 180,E1 -28580.261,E2 -28580.261} C_VEL
LIN {X 0,Y 93.363,Z 893.321,A -85,B 0,C 180,E1 -28582.791,E2 -28582.791} C_VEL
LIN {X 0,Y 98.025,Z 885.743,A -85,B 0,C 180,E1 -28585.177,E2 -28585.177} C_VEL
LIN {X 0,Y 102.37,Z 877.148,A -85,B 0,C 180,E1 -28587.246,E2 -28587.246} C_VEL
LIN {X 0,Y 105.914,Z 868.745,A -85,B 0,C 180,E1 -28588.686,E2 -28588.686} C_VEL
LIN {X 0,Y 109.171,Z 858.999,A -85,B 0,C 180,E1 -28589.865,E2 -28589.865} C_VEL
LIN {X 0,Y 111.828,Z 847.528,A -85,B 0,C 180,E1 -28590.834,E2 -28590.834} C_VEL
LIN {X 0,Y 112.817,Z 839.732,A -85,B 0,C 180,E1 -28591.328,E2 -28591.328} C_VEL
LIN {X 0,Y 111.288,Z 834.65,A -85,B 0,C 180,E1 -28593.512,E2 -28593.512} C_VEL
LIN {X 0,Y 108.32,Z 828.539,A -85,B 0,C 180,E1 -28597.845,E2 -28597.845} C_VEL
LIN {X 0,Y 105.957,Z 823.98,A -85,B 0,C 180,E1 -28602.136,E2 -28602.136} C_VEL
LIN {X 0,Y 103.778,Z 820.096,A -85,B 0,C 180,E1 -28607.417,E2 -28607.417} C_VEL
LIN {X 0,Y 102.248,Z 817.104,A -85,B 0,C 180,E1 -28613.587,E2 -28613.587} C_VEL
LIN {X 0,Y 102.053,Z 815.935,A -85,B 0,C 180,E1 -28615.495,E2 -28615.495} C_VEL
LIN {X 0,Y 101.764,Z 815.458,A -85,B 0,C 180,E1 -28620,E2 -28620} C_VEL
LIN {X 0,Y 102.061,Z 816.143,A -85,B 0,C 180,E1 -28625.186,E2 -28625.186} C_VEL
LIN {X 0,Y 103.173,Z 819.386,A -85,B 0,C 180,E1 -28631.219,E2 -28631.219} C_VEL
LIN {X 0,Y 104.127,Z 820.688,A -85,B 0,C 180,E1 -28634.031,E2 -28634.031} C_VEL
LIN {X 0,Y 106.414,Z 825.061,A -85,B 0,C 180,E1 -28639.283,E2 -28639.283} C_VEL
LIN {X 0,Y 108.643,Z 829.181,A -85,B 0,C 180,E1 -28643.132,E2 -28643.132} C_VEL
LIN {X 0,Y 111.398,Z 834.903,A -85,B 0,C 180,E1 -28647.094,E2 -28647.094} C_VEL
LIN {X 0,Y 112.835,Z 838.495,A -85,B 0,C 180,E1 -28649.084,E2 -28649.084} C_VEL
LIN {X 0,Y 112.645,Z 840.598,A -85,B 0,C 180,E1 -28649.283,E2 -28649.283} C_VEL
LIN {X 0,Y 111.931,Z 844.464,A -85,B 0,C 180,E1 -28649.338,E2 -28649.338} C_VEL
LIN {X 0,Y 110.166,Z 850.115,A -85,B 0,C 180,E1 -28649.209,E2 -28649.209} C_VEL
LIN {X 0,Y 106.15,Z 859.276,A -85,B 0,C 180,E1 -28648.637,E2 -28648.637} C_VEL
LIN {X 0,Y 102.732,Z 866.433,A -85,B 0,C 180,E1 -28648.685,E2 -28648.685} C_VEL
LIN {X 0,Y 101.208,Z 869.895,A -85,B 0,C 180,E1 -28649.082,E2 -28649.082} C_VEL
LIN {X 0,Y 96.558,Z 879.613,A -85,B 0,C 180,E1 -28651.215,E2 -28651.215} C_VEL
LIN {X 0,Y 91.614,Z 887.716,A -85,B 0,C 180,E1 -28653.461,E2 -28653.461} C_VEL
LIN {X 0,Y 86.92,Z 894.396,A -85,B 0,C 180,E1 -28656.044,E2 -28656.044} C_VEL
LIN {X 0,Y 81.703,Z 900.725,A -85,B 0,C 180,E1 -28659.27,E2 -28659.27} C_VEL
LIN {X 0,Y 76.752,Z 905.985,A -85,B 0,C 180,E1 -28662.9,E2 -28662.9} C_VEL
LIN {X 0,Y 72.212,Z 910.372,A -85,B 0,C 180,E1 -28667.057,E2 -28667.057} C_VEL
LIN {X 0,Y 66.159,Z 915.532,A -85,B 0,C 180,E1 -28674.249,E2 -28674.249} C_VEL
LIN {X 0,Y 62.786,Z 918.172,A -85,B 0,C 180,E1 -28679.754,E2 -28679.754} C_VEL
LIN {X 0,Y 58.826,Z 921.063,A -85,B 0,C 180,E1 -28688.997,E2 -28688.997} C_VEL
LIN {X 0,Y 57.039,Z 922.318,A -85,B 0,C 180,E1 -28695.734,E2 -28695.734} C_VEL
LIN {X 0,Y 55.974,Z 923.105,A -85,B 0,C 180,E1 -28702.787,E2 -28702.787} C_VEL
LIN {X 0,Y 55.674,Z 923.404,A -85,B 0,C 180,E1 -28710,E2 -28710} C_VEL
LIN {X 0,Y 55.964,Z 923.123,A -85,B 0,C 180,E1 -28717.214,E2 -28717.214} C_VEL
LIN {X 0,Y 57.023,Z 922.369,A -85,B 0,C 180,E1 -28724.27,E2 -28724.27} C_VEL
LIN {X 0,Y 58.813,Z 921.148,A -85,B 0,C 180,E1 -28731.008,E2 -28731.008} C_VEL
LIN {X 0,Y 62.735,Z 918.294,A -85,B 0,C 180,E1 -28740.273,E2 -28740.273} C_VEL
LIN {X 0,Y 66.103,Z 915.692,A -85,B 0,C 180,E1 -28745.786,E2 -28745.786} C_VEL
LIN {X 0,Y 72.181,Z 910.574,A -85,B 0,C 180,E1 -28752.966,E2 -28752.966} C_VEL
LIN {X 0,Y 77.969,Z 905.065,A -85,B 0,C 180,E1 -28758.043,E2 -28758.043} C_VEL
LIN {X 0,Y 84.224,Z 898.132,A -85,B 0,C 180,E1 -28762.44,E2 -28762.44} C_VEL
LIN {X 0,Y 90.203,Z 890.171,A -85,B 0,C 180,E1 -28765.877,E2 -28765.877} C_VEL
LIN {X 0,Y 95.084,Z 882.576,A -85,B 0,C 180,E1 -28768.213,E2 -28768.213} C_VEL
LIN {X 0,Y 99.503,Z 874.211,A -85,B 0,C 180,E1 -28770.179,E2 -28770.179} C_VEL
LIN {X 0,Y 103.084,Z 865.963,A -85,B 0,C 180,E1 -28771.597,E2 -28771.597} C_VEL
LIN {X 0,Y 106.141,Z 856.896,A -85,B 0,C 180,E1 -28772.791,E2 -28772.791} C_VEL
LIN {X 0,Y 108.694,Z 846.418,A -85,B 0,C 180,E1 -28773.776,E2 -28773.776} C_VEL
LIN {X 0,Y 109.388,Z 841.979,A -85,B 0,C 180,E1 -28774.121,E2 -28774.121} C_VEL
LIN {X 0,Y 107.118,Z 836.042,A -85,B 0,C 180,E1 -28778.165,E2 -28778.165} C_VEL
LIN {X 0,Y 105.04,Z 831.703,A -85,B 0,C 180,E1 -28782.162,E2 -28782.162} C_VEL
LIN {X 0,Y 103.701,Z 829.144,A -85,B 0,C 180,E1 -28785.338,E2 -28785.338} C_VEL
LIN {X 0,Y 102.785,Z 827.04,A -85,B 0,C 180,E1 -28788.163,E2 -28788.163} C_VEL
